	        // write -> global status
	        // Line A1
	        IF #Active.Line.A1 THEN
	            DB_Global.Status.Line.A1.On[#TransferID] := #ReadTransferStatus.ON;
	            DB_Global.Status.Line.A1.ReadyToRun[#TransferID] := #ReadTransferStatus.ReadytoRun;
	            DB_Global.Status.Line.A1.Occupied[#TransferID] := #ReadTransferStatus.Occupied;
	            DB_Global.Status.Line.A1.Running[#TransferID] := #ReadTransferStatus.Running;
	            DB_Global.Status.Line.A1.Fault[#TransferID] := #ReadTransferStatus.Fault;
	            DB_Global.Status.Line.A1.Estop[#TransferID] := #ReadTransferStatus.Estop;
	            DB_Global.Status.Line.A1.Manual[#TransferID] := #ReadTransferStatus.Manual;
	            DB_Global.Status.Line.A1.Stop[#TransferID] := #ReadTransferStatus.Stop;
	            DB_Global.Status.Line.A1.Blockage[#TransferID] := #ReadTransferStatus.Blockage;
	        END_IF;
	        // Line B1
	        IF #Active.Line.B1 THEN
	            DB_Global.Status.Line.B1.On[#TransferID] := #ReadTransferStatus.ON;
	            DB_Global.Status.Line.B1.ReadyToRun[#TransferID] := #ReadTransferStatus.ReadytoRun;
	            DB_Global.Status.Line.B1.Occupied[#TransferID] := #ReadTransferStatus.Occupied;
	            DB_Global.Status.Line.B1.Running[#TransferID] := #ReadTransferStatus.Running;
	            DB_Global.Status.Line.B1.Fault[#TransferID] := #ReadTransferStatus.Fault;
	            DB_Global.Status.Line.B1.Estop[#TransferID] := #ReadTransferStatus.Estop;
	            DB_Global.Status.Line.B1.Manual[#TransferID] := #ReadTransferStatus.Manual;
	            DB_Global.Status.Line.B1.Stop[#TransferID] := #ReadTransferStatus.Stop;
	            DB_Global.Status.Line.B1.Blockage[#TransferID] := #ReadTransferStatus.Blockage;
	        END_IF;
	        // Line C1
	        IF #Active.Line.C1 THEN
	            DB_Global.Status.Line.C1.On[#TransferID] := #ReadTransferStatus.ON;
	            DB_Global.Status.Line.C1.ReadyToRun[#TransferID] := #ReadTransferStatus.ReadytoRun;
	            DB_Global.Status.Line.C1.Occupied[#TransferID] := #ReadTransferStatus.Occupied;
	            DB_Global.Status.Line.C1.Running[#TransferID] := #ReadTransferStatus.Running;
	            DB_Global.Status.Line.C1.Fault[#TransferID] := #ReadTransferStatus.Fault;
	            DB_Global.Status.Line.C1.Estop[#TransferID] := #ReadTransferStatus.Estop;
	            DB_Global.Status.Line.C1.Manual[#TransferID] := #ReadTransferStatus.Manual;
	            DB_Global.Status.Line.C1.Stop[#TransferID] := #ReadTransferStatus.Stop;
	            DB_Global.Status.Line.C1.Blockage[#TransferID] := #ReadTransferStatus.Blockage;
	        END_IF;
	        // Line D1
	        IF #Active.Line.D1 THEN
	            DB_Global.Status.Line.D1.On[#TransferID] := #ReadTransferStatus.ON;
	            DB_Global.Status.Line.D1.ReadyToRun[#TransferID] := #ReadTransferStatus.ReadytoRun;
	            DB_Global.Status.Line.D1.Occupied[#TransferID] := #ReadTransferStatus.Occupied;
	            DB_Global.Status.Line.D1.Running[#TransferID] := #ReadTransferStatus.Running;
	            DB_Global.Status.Line.D1.Fault[#TransferID] := #ReadTransferStatus.Fault;
	            DB_Global.Status.Line.D1.Estop[#TransferID] := #ReadTransferStatus.Estop;
	            DB_Global.Status.Line.D1.Manual[#TransferID] := #ReadTransferStatus.Manual;
	            DB_Global.Status.Line.D1.Stop[#TransferID] := #ReadTransferStatus.Stop;
	            DB_Global.Status.Line.D1.Blockage[#TransferID] := #ReadTransferStatus.Blockage;
	        END_IF;
	        
	    END_REGION
	    
	END_REGION
	
	REGION Transfer Logic
	    
	    REGION infeed receive condition
	        
	        // NegEdgeUpstream
	        #NegEdgeUpstream(CLK := #Upstream);
	        
	        // item will be send into the transfer section when there is no other item
	        
	        IF #ReadTransferStatus.ReadytoRun AND
	            #Upstream AND
	            NOT #ReadTransferStatus.Occupied THEN
	            #Transfer.RcvInfeed := TRUE;
	        END_IF;
	        
	        // receive infeed tag goes to FALSE when the item from the previous conveyor is completly out of the previous conveyor
	        IF NOT #Upstream(* #NegEdgeUpstream.Q *)THEN
	            #Transfer.RcvInfeed := FALSE;
	        END_IF;
	        
	        // Receive infeed
	        #Transfer.StartSignal := #Transfer.RcvInfeed;
	        
	    END_REGION
	    
	    REGION Transfer direction outputs
	        
	        IF NOT #EndSensor AND NOT #"Left/RightSensor" AND NOT #ReadTransferStatus.Running THEN
	            
	            #sTransferDirection := #TransferDirection;
	            
	        END_IF;
	        
	        // Transfer Straight
	        
	        IF #sTransferDirection.Straight THEN
	            
	            IF #ReadTransferStatus.ReadytoRun AND
	                NOT #Transfer.RcvInfeed AND
	                #ReadTransferStatus.Occupied AND
	                NOT #Downstream
	            THEN
	                #Transfer.Command_1 := TRUE;
	                #Transfer.Command_2 := TRUE;
	            END_IF;
	            
	        END_IF;
	        
	        // Transfer Right
	        
	        IF #sTransferDirection.toRight THEN
	            
	            IF #ReadTransferStatus.ReadytoRun AND
	                NOT #Transfer.RcvInfeed AND
	                #ReadTransferStatus.Occupied AND
	                NOT #Downstream
	            THEN
	                #Transfer.Command_1 := TRUE;
	                #Transfer.Command_2 := FALSE;
	            END_IF;
	            
	        END_IF;
	        
	        // Transfer Left
	        
	        IF #sTransferDirection.toLeft THEN
	            
	            IF #ReadTransferStatus.ReadytoRun AND
	                NOT #Transfer.RcvInfeed AND
	                #ReadTransferStatus.Occupied AND
	                NOT #Downstream
	            THEN
	                #Transfer.Command_1 := FALSE;
	                #Transfer.Command_2 := TRUE;
	            END_IF;
	            
	        END_IF;
	        
	    END_REGION
	    
	    REGION TRANSFER OFF
	        
	        // Transfer commands Off
	        
	        IF NOT #ReadTransferStatus.ReadytoRun OR
	            #Transfer.RcvInfeed OR
	            (#ReadTransferStatus.Occupied AND
	            #Downstream) OR
	            NOT #ReadTransferStatus.Occupied
	        THEN
	            #Transfer.Command_1 := FALSE;
	            #Transfer.Command_2 := FALSE;
	        END_IF;
	        
	    END_REGION
	    
	    REGION Write output
	        
	        // Static to output
	        
	        #StartSignal := #Transfer.StartSignal;
	        #Cmd1 := #Transfer.Command_1;
	        #Cmd2 := #Transfer.Command_2;
	        
	    END_REGION
	    
	END_REGION
	
	
	
	
	
END_FUNCTION_BLOCK
END_NAMESPACE

NAMESPACE LineA1
FUNCTION_BLOCK FB_GetDiag
{ S7_Optimized_Access := 'TRUE' ; Published := 'TRUE' }
VERSION : 0.1
   VAR_INPUT 
      HardwareID : HW_ANY;
   END_VAR

   VAR_OUTPUT 
      CommunicationErrorAlarm : Bool;
   END_VAR

   VAR 
      GetDiag { S7_SetPoint := 'False'} : _.Global.GetDiag;
      CheckOwnState : UInt := 5;
      CommunicationError : Bool;
   END_VAR


BEGIN
	// ==========================================================================================================================================
	// Company        : LogTech, s.r.o.
	// Created by     : Anton Vinoth Soundraraj
	// Block          : FB_GetDiag
	// Project        : LT-Lib-Block
	// ==========================================================================================================================================
	
	REGION Get_Diag
	    
	    #GetDiag.ReturnValue := GET_DIAG(MODE := #GetDiag.DiagMode,
	                                     LADDR := #HardwareID,
	                                     CNT_DIAG => #GetDiag.CountDiagDetail,
	                                     DIAG := #GetDiag.MyDiag);
	END_REGION
	
	REGION Communiation_Error
	    
	    IF #GetDiag.MyDiag.OwnState = #CheckOwnState THEN
	        #CommunicationErrorAlarm := TRUE;
	    ELSE
	        #CommunicationErrorAlarm := FALSE;
	    END_IF;
	    
	    IF #GetDiag.MyDiag.OwnState = #CheckOwnState THEN
	        #CommunicationError := TRUE;
	    ELSE
	        #CommunicationError := FALSE;
	    END_IF;
	    
	END_REGION
	
	
END_FUNCTION_BLOCK
END_NAMESPACE

NAMESPACE Global
FUNCTION_BLOCK FB_HardwareDiag
{ S7_Optimized_Access := 'TRUE' ; Published := 'TRUE' }
VERSION : 0.1
   VAR 
      ASi : _.LineA1.FB_GetDiag;
   END_VAR


BEGIN
	// ==========================================================================================================================================
	// Company        : LogTech, s.r.o.
	// Created by     : Anton Vinoth Soundraraj
	// Block          : FB_HardwareDiag
	// Project        : Lékarna DC Chrudim
	// Project number : 23-157
	// ==========================================================================================================================================
	
	(* REGION ASi
	    
	    #ASi(HardwareID              := _."bu-asi-gw~PN-IO",
	         CommunicationErrorAlarm => _.Global.DB_Alarm.HardDiag.ASi.%X0);
	    
	    
	END_REGION *)
	
	
	
	
END_FUNCTION_BLOCK
END_NAMESPACE

NAMESPACE Global
FUNCTION FC_AllKlaxon : Void
{ S7_Optimized_Access := 'TRUE' ; Published := 'TRUE' }
VERSION : 0.1

BEGIN
	// ==========================================================================================================================================
	// Company        : LogTech, s.r.o.
	// Created by     : Anton Vinoth Soundraraj
	// Block          : FB_HardwareDiag
	// Project        : Lékarna DC Chrudim
	// Project number : 23-157
	// ==========================================================================================================================================
	
	
END_FUNCTION
END_NAMESPACE

NAMESPACE LineA1
FUNCTION FC_Init : Void
{ S7_Optimized_Access := 'TRUE' ; Published := 'TRUE' }
VERSION : 0.1

BEGIN
	
	
	
	_.LineA1.IDB_LineA1."Conveyor_A1.1.1".MotorType."24v-ASi" := TRUE;
	
	
	
	
	
	
	
	
	
	
	
	
	
	
END_FUNCTION
END_NAMESPACE

NAMESPACE LineA1
FUNCTION_BLOCK FB_Interlock
{ S7_Optimized_Access := 'TRUE' ; Published := 'TRUE' }
VERSION : 0.1

BEGIN
END_FUNCTION_BLOCK
END_NAMESPACE

NAMESPACE LineA1
FUNCTION FC_Downstream : Void
{ S7_Optimized_Access := 'TRUE' ; Published := 'TRUE' }
VERSION : 0.1

BEGIN
END_FUNCTION
END_NAMESPACE

NAMESPACE LineA1
FUNCTION FC_Fault : Void
{ S7_Optimized_Access := 'TRUE' ; Published := 'TRUE' }
VERSION : 0.1

BEGIN
END_FUNCTION
END_NAMESPACE

NAMESPACE LineA1
FUNCTION FC_Upstream : Void
{ S7_Optimized_Access := 'TRUE' ; Published := 'TRUE' }
VERSION : 0.1

BEGIN
END_FUNCTION
END_NAMESPACE

NAMESPACE LineA1
FUNCTION FC_Alarm : Void
{ S7_Optimized_Access := 'TRUE' ; Published := 'TRUE' }
VERSION : 0.1

BEGIN
END_FUNCTION
END_NAMESPACE

NAMESPACE LineA1
FUNCTION FC_SimuAlarm : Void
{ S7_Optimized_Access := 'TRUE' ; Published := 'FALSE' }
VERSION : 0.1

BEGIN
END_FUNCTION
END_NAMESPACE

NAMESPACE LineB1
FUNCTION_BLOCK FB_S300_FullControl
{ S7_Optimized_Access := 'TRUE' ; Published := 'TRUE' }
VERSION : 0.1
   VAR_INPUT 
      TransferID : Int;
      TransferSensor : Bool;
      BeltUp : Bool;
      RollerUp : Bool;
      Fault : Bool;
      ReadyToRCV : Bool;
      UpstreamStraight : Bool;
      UpstreamArm : Bool;
      FrontSensor : Bool;
      EndSensor : Bool;
      "Left/RightSensor" : Bool;
      Downstream : Bool;
      PriorityStraight : Bool;
      PriorityArm : Bool;
      FrontSensorFilterTime : Array[1..2] of Time;
   END_VAR

   VAR_OUTPUT 
      Direction : Bool;
      Cmd1 : Bool;
      Cmd2 : Bool;
      ErrorReset : Bool;
   END_VAR

   VAR 
      ReadInputSignal : Struct
         EmergencyStop : Bool;
         FireActive : Bool;
         Fault : Bool;
         TransferSensor : Bool;
      END_STRUCT;
      Active : Struct
         Line : Struct
            B1 : Bool;
         END_STRUCT;
      END_STRUCT;
      TRANSFER_SENSOR : _.Global.FB_Sensor;
      FRONT_SENSOR_FILTER : _.Global.FB_Sensor;
      TRANSFER_SENSOR_BLOCKAGE {InstructionName := 'TON_TIME'; LibVersion := '1.0'} : TON_TIME;
      FRONT_SENSOR_BLOCKAGE {InstructionName := 'TON_TIME'; LibVersion := '1.0'} : TON_TIME;
      END_SENSOR_BLOCKAGE {InstructionName := 'TON_TIME'; LibVersion := '1.0'} : TON_TIME;
      "LEFT/RIGHT_SENSOR_BLOCKAGE" {InstructionName := 'TON_TIME'; LibVersion := '1.0'} : TON_TIME;
      TRANSFER_STATUS_ON : _.Global.FB_StatusON;
      TRANSFER_STATUS_READY : _.Global.FB_StatusReady;
      TRANSFER_STATUS_FAULT : _.Global.FB_StatusFault;
      AUTO_RESET : _.Global.FB_AutoReset;
      StartUpTimer {InstructionName := 'TOF_TIME'; LibVersion := '1.0'; S7_SetPoint := 'False'} : TOF_TIME;
      FT_StartUp {InstructionName := 'F_TRIG'; LibVersion := '1.0'} : F_TRIG;
      SetStartUp { S7_SetPoint := 'True'} : Bool;
      Init : Struct
         Line : Struct
            A1 : String := 'LineA1';
         END_STRUCT;
      END_STRUCT;
      SSR : _.Global.SystemSSR;
      ReadTransferStatus : _.Global.ConveyorStatus;
      ReadTransferParameters : _.Global.ConveyorParameters := ((), [2(T#10ms)], (), (), ());
      ConveyorFault : _.Global.Fault;
      StartupTransfer { S7_SetPoint := 'True'} : Bool;
      FilteredSensor { S7_SetPoint := 'True'} : Bool;
      StopSystemFireActive : Bool;
      ClearTransferArea : Bool;
      AutoReset : Bool;
      VisuColor : Word;
      Transfer : Struct
         ErrorReset : Bool;
         Direction : Bool;
         Command_1 : Bool;
         Command_2 : Bool;
      END_STRUCT;
   END_VAR


BEGIN
	// ==========================================================================================================================================
	// Company        : LogTech, s.r.o.
	// Created by     : Anton Vinoth Soundraraj
	// Block          : FB_S300_tTransMode
	// Project        : Lékarna DC Chrudim
	// Project number : 23-157
	// ==========================================================================================================================================
	
	REGION Active Line
	    
	        #Active.Line.B1 := TRUE;
	        
	END_REGION
	
	REGION SystemSSR
	    
	    // Line B1
	    IF #Active.Line.B1 THEN
	        #SSR.StartSystem := _.Global.DB_SystemSSR.Line.B1.StartSystem;
	        #SSR.StopSystem := _.Global.DB_SystemSSR.Line.B1.StopSystem;
	        #SSR.ResetSystem := _.Global.DB_SystemSSR.Line.B1.ResetSystem;
	    END_IF;
	    
	END_REGION
	
	REGION Read Input
	    
	    // read all inputs to the block
	    // Conveyor input read signals
	    #ReadInputSignal.TransferSensor := #TransferSensor;
	    #ReadInputSignal.Fault := #Fault;
	    // Read static tag connections
	    #ReadInputSignal.EmergencyStop := // all estop zones are connected together
	    _.DB_SafetyStandard.ToStandard.EstopActive;
	    // Common system input Read
	    #ReadInputSignal.FireActive :=
	    _.Global.DB_SystemSimu.Fire; // simu call
	    
	END_REGION
	
	REGION Conveyor startup
	    
	    // Conveyor StartUp: Conveyor startup signal after preset time
	    #StartUpTimer.TOF(IN := #SSR.StartSystem,
	                      PT := #ReadTransferParameters.StartUpTime);
	    
	    #FT_StartUp(CLK := #StartUpTimer.Q);
	    
	    // set startup after the preset
	    #SetStartUp := #FT_StartUp.Q;
	    
	END_REGION
	
	REGION READ AND INIT
	    
	    REGION Init conveyor parameters
	        
	        // Conveyor Parameter
	        // Line B1
	        IF #Active.Line.B1 THEN
	            #ReadTransferParameters := DB_ConveyorParameters.Line.B1.Conveyor[#TransferID];
	        END_IF;
	        
	    END_REGION
	    
	    REGION Sensor Filter
	        
	        // FB_Sensor
	        // called as MIDB
	        
	        #TRANSFER_SENSOR(Sensor := #ReadInputSignal.TransferSensor,
	                         SensorFilterTime := #ReadTransferParameters.SensorFilterTime,
	                         FilteredSensor => #FilteredSensor);
	        
	        // front sensor filter
	        #FRONT_SENSOR_FILTER(Sensor := #FrontSensor,
	                             SensorFilterTime := #FrontSensorFilterTime);
	        
	    END_REGION
	    
	    REGION FIRE
	        
	        // Fire signal from fire system stops the whole system
	        // System can be reset from Fire status only if the fire signal is deactivated
	        
	        // FIRE ALARM ACTIVE --> STOP SYSTEM
	        IF #ReadInputSignal.FireActive THEN
	            #StopSystemFireActive := TRUE;
	        END_IF;
	        // RESET --> FIRE ALARM
	        IF #SSR.ResetSystem AND NOT #ReadInputSignal.FireActive THEN
	            #StopSystemFireActive := FALSE;
	        END_IF;
	        
	    END_REGION
	    
	END_REGION
	
	REGION Conveyor Status
	    
	    REGION Status ON
	        
	        // ----------------------------------------->>>>>>> STATUS ON <<<<<<<-----------------------------------------
	        // FB_ConveyorStatusON
	        // called as IDMB
	        
	        #TRANSFER_STATUS_ON(SystemStartActive := #SSR.StartSystem,
	                            StatusStop := #ReadTransferStatus.Stop,
	                            StatusEStop := #ReadTransferStatus.Estop,
	                            StatusManual := #ReadTransferStatus.Manual,
	                            StatusFault := #ReadTransferStatus.Fault,
	                            FireAlarmActive := #StopSystemFireActive,
	                            StatusON => #ReadTransferStatus.ON);
	        
	    END_REGION
	    
	    REGION Status Ready
	        
	        // ----------------------------------------->>>>>>> STATUS READY <<<<<<<-----------------------------------------
	        // FB_ConveyorStatusReady
	        // called as MIDB
	        
	        #TRANSFER_STATUS_READY(StatusON := #ReadTransferStatus.ON,
	                               StatusESTOP := #ReadTransferStatus.Estop,
	                               StatusFAULT := #ReadTransferStatus.Fault,
	                               StatusMAN := #ReadTransferStatus.Manual,
	                               SignalFIRE := #StopSystemFireActive,
	                               SystemAlertTime := #ReadTransferParameters.StartUpTime,
	                               StatusReady => #ReadTransferStatus.ReadytoRun);
	        
	    END_REGION
	    
	    REGION Status Occupied
	        
	        // ----------------------------------------->>>>>>> STATUS OCCUPIED <<<<<<<-----------------------------------------
	        
	        #ReadTransferStatus.Occupied :=
	        #FilteredSensor AND
	        NOT #FRONT_SENSOR_FILTER.FilteredSensor;
	        
	    END_REGION
	    
	    REGION Status Running
	        
	        // ----------------------------------------->>>>>>> STATUS RUNNING <<<<<<<-----------------------------------------
	        
	        #ReadTransferStatus.Running := #Transfer.Command_1 OR #Transfer.Command_2;
	        
	    END_REGION
	    
	    REGION Status Fault
	        
	        // Automatic reset trigger to the needed drive after wakeup from ESTOP power miss (only if needed)
	        // will trigger for every Reset active
	        
	        #AUTO_RESET(AckIN := #SSR.ResetSystem,
	                    Ack => #AutoReset);
	        
	        // ----------------------------------------->>>>>>> STATUS FAULT <<<<<<<-----------------------------------------
	        
	        #TRANSFER_STATUS_FAULT(FaultActive := #ReadInputSignal.Fault,
	                               ResetFault := #SSR.ResetSystem OR #AutoReset,
	                               StatusRunning := #ReadTransferStatus.Running,
	                               FaultStatus => #ReadTransferStatus.Fault);
	        
	        #ErrorReset := #SSR.ResetSystem AND #ReadTransferStatus.Fault;
	        
	    END_REGION
	    
	    REGION Status ESTOP
	        
	        // ----------------------------------------->>>>>>> STATUS ESTOP <<<<<<<-----------------------------------------
	        
	        // EMERGENCY STOP ACTIVE --> STOP SYSTEM
	        IF #ReadInputSignal.EmergencyStop THEN
	            #ReadTransferStatus.Estop := TRUE;
	        END_IF;
	        // RESET --> EMERGENCY STOP
	        IF #AutoReset AND NOT #ReadInputSignal.EmergencyStop THEN
	            #ReadTransferStatus.Estop := FALSE;
	        END_IF;
	        
	    END_REGION
	    
	    REGION Status Manual
	        
	        // ----------------------------------------->>>>>>> STATUS MANUAL <<<<<<<-----------------------------------------
	        
	        // Write to static from IO
	        // ACTIVATE --> MANUAL MODE
	        // Line B1
	        IF #Active.Line.B1 THEN
	            // SET --> MANUAL MODE
	            IF DB_Manual.Line.B1.Conveyor[#TransferID].ManualEnable THEN
	                #ReadTransferStatus.Manual := TRUE;
	            END_IF;
	            // RESET --> MANUAL MODE
	            IF NOT DB_Manual.Line.B1.Conveyor[#TransferID].ManualEnable AND #SSR.ResetSystem THEN
	                #ReadTransferStatus.Manual := FALSE;
	            END_IF;
	        END_IF;
	        
	    END_REGION
	    
	    REGION Status Stop
	        
	        // ----------------------------------------->>>>>>> STATUS STOP <<<<<<<-----------------------------------------
	        
	        IF #SSR.StopSystem THEN
	            #ReadTransferStatus.Stop := TRUE;
	        END_IF;
	        IF #SSR.StartSystem OR #SSR.ResetSystem THEN
	            #ReadTransferStatus.Stop := FALSE;
	        END_IF;
	        
	    END_REGION
	    
	    REGION Status Blockage
	        
	        // FB_SensorBlockage
	        // called as MIDB
	        #TRANSFER_SENSOR_BLOCKAGE(IN := #ReadTransferStatus.ReadytoRun AND #FilteredSensor AND NOT #Downstream,
	                                  PT := T#15s);
	        
	        #FRONT_SENSOR_BLOCKAGE(IN := #ReadTransferStatus.ReadytoRun AND #FrontSensor AND NOT #Downstream,
	                               PT := T#15s);
	        
	        #END_SENSOR_BLOCKAGE(IN := #ReadTransferStatus.ReadytoRun AND #EndSensor AND NOT #Downstream,
	                             PT := T#15s);
	        
	        #"LEFT/RIGHT_SENSOR_BLOCKAGE"(IN := #ReadTransferStatus.ReadytoRun AND #"Left/RightSensor" AND NOT #Downstream,
	                                      PT := T#5s);
	        
	        #ReadTransferStatus.Blockage :=
	        (#TRANSFER_SENSOR_BLOCKAGE.Q OR
	        #FRONT_SENSOR_BLOCKAGE.Q OR
	        #END_SENSOR_BLOCKAGE.Q OR
	        #"LEFT/RIGHT_SENSOR_BLOCKAGE".Q);
	        
	        // ==========================
	        // Sensor Blockage: HMI Alarm
	        // ==========================
	        // Sensor blockage alarm message is written to the alarm word
	        // corresponding to the active line
	        
	        REGION alarm 
	            
	            // ==========================
	            // Sensor Blockage: HMI Alarm
	            // ==========================
	            // Sensor blockage alarm message is written to the alarm word
	            // corresponding to the active line
	            // Line B1
	            IF #Active.Line.B1 THEN
	                DB_Alarm."word".Line.B1.Conveyor[#TransferID].%X0 := #ReadTransferStatus.Blockage;
	            END_IF;
	            
	        END_REGION
	        
	    END_REGION
	    
	    REGION Visu Color
	        
	        // each and every status of the conveyor will be mentioned by different colors in HMI panel
	        
	        #VisuColor.%X8 := #ReadTransferStatus.Blockage;
	        #VisuColor.%X0 := #ReadTransferStatus.ON;
	        #VisuColor.%X1 := #ReadTransferStatus.ReadytoRun;
	        #VisuColor.%X2 := #ReadTransferStatus.Occupied;
	        #VisuColor.%X3 := #ReadTransferStatus.Running;
	        #VisuColor.%X4 := #ReadTransferStatus.Fault;
	        #VisuColor.%X5 := #ReadTransferStatus.Estop;
	        #VisuColor.%X6 := #ReadTransferStatus.Manual;
	        #VisuColor.%X7 := #ReadTransferStatus.Stop;
	        
	        // convert word to Interger value: 
	        // color will be depends on the status priority (integer value) 
	        // reference: Conveyor image in HMI screen -> property -> Apperance   
	        
	        // Line B1
	        IF #Active.Line.B1 THEN
	            _.Global.DB_VisuColor.Line.B1.Conveyor[#TransferID] :=
	            WORD_TO_INT(#VisuColor);
	        END_IF;
	        
	    END_REGION
	    
	    REGION Global Status
	        
	        // write -> global status
	        // Line B1
	        IF #Active.Line.B1 THEN
	            _.Global.DB_Global.Status.Line.B1.On[#TransferID] := #ReadTransferStatus.ON;
	            _.Global.DB_Global.Status.Line.B1.ReadyToRun[#TransferID] := #ReadTransferStatus.ReadytoRun;
	            _.Global.DB_Global.Status.Line.B1.Occupied[#TransferID] := #ReadTransferStatus.Occupied;
	            _.Global.DB_Global.Status.Line.B1.Running[#TransferID] := #ReadTransferStatus.Running;
	            _.Global.DB_Global.Status.Line.B1.Fault[#TransferID] := #ReadTransferStatus.Fault;
	            _.Global.DB_Global.Status.Line.B1.Estop[#TransferID] := #ReadTransferStatus.Estop;
	            _.Global.DB_Global.Status.Line.B1.Manual[#TransferID] := #ReadTransferStatus.Manual;
	            _.Global.DB_Global.Status.Line.B1.Stop[#TransferID] := #ReadTransferStatus.Stop;
	            _.Global.DB_Global.Status.Line.B1.Blockage[#TransferID] := #ReadTransferStatus.Blockage;
	        END_IF;
	        
	    END_REGION
	    
	END_REGION
	
	REGION Transfer Logic
	    
	    IF #ReadTransferStatus.ReadytoRun THEN
	        
	        REGION Belt going UP
	            
	            // tote from straight has higher priority
	            // upstream straight is satisfied (add upstream sensor and front sensor)
	            // transfer is not occupied
	            // belt is not UP
	            IF (#PriorityStraight AND
	                #UpstreamStraight AND
	                NOT #ReadTransferStatus.Occupied AND
	                NOT #BeltUp) OR
	                // transfer has received an item from arm
	                // belt is not UP
	                (#ReadTransferStatus.Occupied AND
	                NOT #BeltUp)
	            THEN
	                #Transfer.Command_1 := TRUE;
	                #Transfer.Command_2 := TRUE;
	                #Transfer.Direction := TRUE;
	            END_IF;
	            
	        END_REGION
	        
	        REGION Roller going UP
	            
	            // tote from arm has higher priority
	            // upstream arm is satisfied (add upstream sensor and left/right sensor)
	            // transfer is not occupied
	            // roller is not UP
	            IF (#PriorityArm AND
	                #UpstreamArm AND
	                NOT #ReadTransferStatus.Occupied AND
	                NOT #RollerUp)
	            THEN
	                #Transfer.Command_1 := TRUE;
	                #Transfer.Command_2 := TRUE;
	                #Transfer.Direction := FALSE;
	            END_IF;
	            
	        END_REGION
	        
	        REGION Belt rcv and trs item
	            
	            IF // belt rcv the item (from straight)
	                (#BeltUp AND
	                NOT #ReadTransferStatus.Occupied AND
	                #PriorityStraight AND
	                #UpstreamStraight) OR
	                // belt trs the item
	                (#BeltUp AND
	                #ReadTransferStatus.Occupied AND
	                NOT #Downstream)
	            THEN
	                #Transfer.Command_1 := TRUE;
	                #Transfer.Command_2 := FALSE;
	                #Transfer.Direction := FALSE;
	            END_IF;
	            
	        END_REGION
	        
	    END_IF;
	    
	    REGION TRANSFER OFF
	        
	        IF NOT #ReadTransferStatus.ReadytoRun OR
	            (#ReadTransferStatus.Occupied AND
	            #Downstream)
	        THEN
	            #Transfer.Command_1 := FALSE;
	            #Transfer.Command_2 := FALSE;
	        END_IF;
	        
	    END_REGION
	    
	    REGION Write output
	        
	        // Static to output
	        
	        #Direction := #Transfer.Direction;
	        #Cmd1 := #Transfer.Command_1;
	        #Cmd2 := #Transfer.Command_2;
	        #ErrorReset := #Transfer.ErrorReset;
	        
	    END_REGION
	    
	END_REGION
	
	
	
	
	
END_FUNCTION_BLOCK
END_NAMESPACE

NAMESPACE Global
FUNCTION_BLOCK FB_MABS_Profinet
{ S7_Optimized_Access := 'TRUE' ; Published := 'TRUE' }
VERSION : 0.1
   VAR_INPUT 
      MABS_ID : Int;
      CrossSensor : Bool;
      Fault : Bool;
      UpstreamRunning : Bool;
      Downstream_Straight : Bool;
      "Downstream_Right/Left" : Bool;
      SortDir : ItemDir;
      ManIn : MABS_ManIn;
      Setpoints : MABS_Setpoint;
   END_VAR

   VAR_IN_OUT 
      MABS_IBP_in : IB_P01_02_03_in_64bytes_struct;
      MABS_IBP_out : IB_P01_02_03_out_64bytes_struct;
   END_VAR

   VAR 
      ReadInputSignal : Struct
         CrossSensor : Bool;
         EmergencyStop : Bool;
         Fault : Bool;
      END_STRUCT;
      Active : Struct
         Line : Struct
            ProductionLine : Bool;
            EmptyLine : Bool;
            PackedLine : Bool;
         END_STRUCT;
         EstopZone { S7_SetPoint := 'False'} : EsopZone;
      END_STRUCT;
      CROSS_SENSOR_FILTER : FB_Sensor;
      MABS_SENSOR_BLOCKAGE {InstructionName := 'IEC_TIMER'; LibVersion := '1.0'} : IEC_TIMER;
      MABS_STATUS_ON : FB_StatusON;
      MABS_STATUS_READY : FB_StatusReady;
      MABS_STATUS_FAULT : FB_StatusFault;
      AUTO_RESET : FB_AutoReset;
      MABS_CONTROL : FB_MABS_PNIO;
      SSR : SystemSSR;
      ReadMabsStatus : ConveyorStatus;
      ReadMabsParameter : ConveyorParameters := ((), [2(T#10ms)], (), (), (), ());
      MABSFault : Fault;
      SimuMode : Struct
         Sensor : Bool;
         Fault : Bool;
      END_STRUCT;
      StartUpTimer {InstructionName := 'TOF_TIME'; LibVersion := '1.0'; S7_SetPoint := 'False'} : TOF_TIME;
      FT_StartUp {InstructionName := 'F_TRIG'; LibVersion := '1.0'} : F_TRIG;
      SetStartUp { S7_SetPoint := 'True'} : Bool;
      VisuColor : Word;
      PhaseError : Bool;
      StartupMABS { S7_SetPoint := 'True'} : Bool;
      FilteredSensor { S7_SetPoint := 'True'} : Bool;
      AutoReset { S7_SetPoint := 'True'} : Bool;
      StopSystemFireActive : Bool;
      Sort { S7_SetPoint := 'False'} : ItemDir;
      Home : Bool;
      HomeCheckTimer {InstructionName := 'TON_TIME'; LibVersion := '1.0'} : TON_TIME;
      CurrentPosition : Struct
         left : Bool;
         right : Bool;
         straight : Bool;
      END_STRUCT;
      "Cmd+Setpoint" { ExternalAccessible := 'False'; ExternalVisible := 'False'; ExternalWritable := 'False'; S7_SetPoint := 'False'} : MABS;
   END_VAR


BEGIN
	// ==========================================================================================================================================
	// Company        : LogTech, s.r.o.
	// Created by     : Anton Vinoth Soundraraj
	// Block          : FB_MABS
	// Project        : Lékarna DC Chrudim
	// Project number : 23-157
	// ==========================================================================================================================================
	
	REGION Active Line
	    
	    // ProductionLine
	    IF (#MABS_ID >= _.gminProductionLine AND
	        #MABS_ID <= _.gmaxProductionLine)
	    THEN
	        #Active.Line.ProductionLine := TRUE;
	    END_IF;
	    
	    // EmptyLine
	    IF (#MABS_ID >= _.gminEmptyLine AND
	        #MABS_ID <= _.gmaxEmptyLine)
	    THEN
	        #Active.Line.EmptyLine := TRUE;
	    END_IF;
	    
	    // PackedLine
	    IF (#MABS_ID >= _.gminPackedLine AND
	        #MABS_ID <= _.gmaxPackedLine)
	    THEN
	        #Active.Line.PackedLine := TRUE;
	    END_IF;
	    
	END_REGION
	
	REGION Estop zone
	    
	    // Production Line A1
	    IF  (#MABS_ID >= _."gA1.6.1" AND
	        #MABS_ID <= _."gA1.6.2") OR
	        // Empty Line A1
	        (#MABS_ID >= _."gJ1.5.2" AND
	        #MABS_ID <= _."gJ1.6.2")
	    THEN
	        #Active.EstopZone."1" := TRUE;
	    END_IF;
	    
	    // Production Line A2
	    IF  (#MABS_ID >= _."gA1.9.1" AND
	        #MABS_ID <= _."gA1.9.2")
	    THEN
	        #Active.EstopZone."2" := TRUE;
	    END_IF;
	    
	END_REGION
	
	REGION SystemSSR
	    
	    //Zone 1
	    IF #Active.EstopZone."1" THEN
	        #SSR.StartSystem := DB_SystemSSR.Zone."1".StartSystem;
	        #SSR.StopSystem := DB_SystemSSR.Zone."1".StopSystem;
	        #SSR.ResetSystem := DB_SystemSSR.Zone."1".ResetSystem;
	    END_IF;
	    
	    //Zone 2
	    IF #Active.EstopZone."2" THEN
	        #SSR.StartSystem := DB_SystemSSR.Zone."2".StartSystem;
	        #SSR.StopSystem := DB_SystemSSR.Zone."2".StopSystem;
	        #SSR.ResetSystem := DB_SystemSSR.Zone."2".ResetSystem;
	    END_IF;
	    
	END_REGION
	
	REGION Read Simu inputs  
	    
	    // ProductionLine
	    IF #Active.Line.ProductionLine THEN
	        // read simu
	        #SimuMode.Sensor := DB_SystemSimu.TriggerSensor.Line.ProductionLine.Conveyor[#MABS_ID];
	        #SimuMode.Fault := DB_SystemSimu.TriggerFault.Line.ProductionLine.Conveyor[#MABS_ID];
	    END_IF;
	    
	    // EmptyLine
	    IF #Active.Line.EmptyLine THEN
	        // read simu
	        #SimuMode.Sensor := DB_SystemSimu.TriggerSensor.Line.EmptyLine.Conveyor[#MABS_ID];
	        #SimuMode.Fault := DB_SystemSimu.TriggerFault.Line.EmptyLine.Conveyor[#MABS_ID];
	    END_IF;
	    
	    // PackedLine
	    IF #Active.Line.PackedLine THEN
	        // read simu
	        #SimuMode.Sensor := DB_SystemSimu.TriggerSensor.Line.PackedLine.Conveyor[#MABS_ID];
	        #SimuMode.Fault := DB_SystemSimu.TriggerFault.Line.PackedLine.Conveyor[#MABS_ID];
	    END_IF;
	    
	END_REGION
	
	REGION Read Input
	    
	    // read all inputs to the block
	    // Conveyor input read signals
	    #ReadInputSignal.CrossSensor := #CrossSensor OR  // Not
	    #SimuMode.Sensor; // simu call
	    #ReadInputSignal.Fault := #Fault OR
	    #SimuMode.Fault; // simu call;
	    #ReadInputSignal.EmergencyStop := // all estop zones are connected together
	    _.DB_SafetyStandard.ToStandard.EstopActive;
	    
	END_REGION
	
	REGION READ AND INIT
	    
	    REGION parameters
	        
	        // ProductionLine
	        IF #Active.Line.ProductionLine THEN
	            #ReadMabsParameter := DB_ConveyorParameters.Line.ProductionLine.Conveyor[#MABS_ID];
	        END_IF;
	        // EmptyLine
	        IF #Active.Line.EmptyLine THEN
	            #ReadMabsParameter := DB_ConveyorParameters.Line.EmptyLine.Conveyor[#MABS_ID];
	        END_IF;
	        // PackedLine
	        IF #Active.Line.PackedLine THEN
	            #ReadMabsParameter := DB_ConveyorParameters.Line.PackedLine.Conveyor[#MABS_ID];
	        END_IF;
	        
	    END_REGION
	    
	    REGION FIRE
	        
	        // Fire signal from fire system stops the whole system
	        // System can be reset from Fire status only if the fire signal is deactivated
	        
	        // FIRE ALARM ACTIVE --> STOP SYSTEM
	        IF DB_SystemSimu.Fire THEN
	            #StopSystemFireActive := TRUE;
	        END_IF;
	        // RESET --> FIRE ALARM
	        IF #SSR.ResetSystem AND NOT DB_SystemSimu.Fire THEN
	            #StopSystemFireActive := FALSE;
	        END_IF;
	        
	    END_REGION
	    
	END_REGION
	
	REGION Conveyor startup
	    
	    // Conveyor StartUp: Conveyor startup signal after 5 second delay
	    
	    #StartUpTimer.TOF(IN := #SSR.StartSystem,
	                      PT := #ReadMabsParameter.StartUpTime);
	    
	    #FT_StartUp(CLK := #StartUpTimer.Q);
	    
	    // set startup after 5 seconds
	    #SetStartUp := #FT_StartUp.Q;
	    
	END_REGION
	
	REGION Conveyor Status
	    
	    REGION Status ON
	        
	        // ----------------------------------------->>>>>>> STATUS ON <<<<<<<-----------------------------------------
	        // FB_ConveyorStatusON
	        // called as IDMB
	        
	        #MABS_STATUS_ON(SystemStartActive := #SSR.StartSystem,
	                        StatusStop := #ReadMabsStatus.Stop,
	                        StatusEStop := #ReadMabsStatus.Estop,
	                        StatusManual := #ReadMabsStatus.Manual,
	                        StatusFault := #ReadMabsStatus.Fault,
	                        FireAlarmActive := #StopSystemFireActive,
	                        StatusON => #ReadMabsStatus.ON);
	        
	    END_REGION
	    
	    REGION Status Ready
	        
	        // ----------------------------------------->>>>>>> STATUS READY <<<<<<<-----------------------------------------
	        // FB_ConveyorStatusReady
	        // called as MIDB
	        
	        #MABS_STATUS_READY(StatusON := #ReadMabsStatus.ON,
	                           StatusESTOP := #ReadMabsStatus.Estop,
	                           StatusFAULT := #ReadMabsStatus.Fault,
	                           StatusMAN := #ReadMabsStatus.Manual,
	                           SignalFIRE := #StopSystemFireActive,
	                           SystemAlertTime := #ReadMabsParameter.StartUpTime,
	                           StatusReady => #ReadMabsStatus.ReadytoRun);
	        
	    END_REGION
	    
	    REGION Status Occupied
	        
	        // ----------------------------------------->>>>>>> STATUS OCCUPIED <<<<<<<-----------------------------------------
	        
	        #ReadMabsStatus.Occupied :=
	        #CROSS_SENSOR_FILTER.FilteredSensor;
	        
	    END_REGION
	    
	    REGION Status Running
	        
	        // ----------------------------------------->>>>>>> STATUS RUNNING <<<<<<<-----------------------------------------
	        
	        #ReadMabsStatus.Running :=
	        #ReadMabsStatus.ReadytoRun AND
	        #"Cmd+Setpoint".Run_balls;
	        
	    END_REGION
	    
	    REGION Status Fault
	        
	        // ----------------------------------------->>>>>>> STATUS FAULT <<<<<<<-----------------------------------------
	        
	        // Reading error signal from the motor drive
	        #MABSFault.Motor_Error := #ReadInputSignal.Fault;
	        
	        // FC_ConveyorStatusFault
	        #MABS_STATUS_FAULT(FaultActive := #MABSFault.Motor_Error,
	                           ResetFault := #SSR.ResetSystem,
	                           StatusRunning := #ReadMabsStatus.Running,
	                           FaultStatus => #ReadMabsStatus.Fault);
	        
	    END_REGION
	    
	    REGION Status ESTOP
	        
	        // ----------------------------------------->>>>>>> STATUS ESTOP <<<<<<<-----------------------------------------
	        
	        #AUTO_RESET(AckIN := #SSR.ResetSystem,
	                    Ack => #AutoReset);
	        
	        // EMERGENCY STOP ACTIVE --> STOP SYSTEM
	        IF #ReadInputSignal.EmergencyStop THEN
	            #ReadMabsStatus.Estop := TRUE;
	        END_IF;
	        // RESET --> EMERGENCY STOP
	        IF #AutoReset AND NOT #ReadInputSignal.EmergencyStop THEN
	            #ReadMabsStatus.Estop := FALSE;
	        END_IF;
	        
	    END_REGION
	    
	    REGION Status Stop
	        
	        // ----------------------------------------->>>>>>> STATUS STOP <<<<<<<-----------------------------------------
	        
	        IF #SSR.StopSystem THEN
	            #ReadMabsStatus.Stop := TRUE;
	        END_IF;
	        IF #SSR.StartSystem OR #SSR.ResetSystem THEN
	            #ReadMabsStatus.Stop := FALSE;
	        END_IF;
	        
	    END_REGION
	    
	    REGION Sensor Blockage
	        
	        // ----------------------------------------->>>>>>> STATUS BLOCKAGE <<<<<<<-------------------------------------
	        
	        // FB_SensorBlockage
	        // called as MIDB
	        
	        #MABS_SENSOR_BLOCKAGE.TON(IN := #ReadMabsStatus.ReadytoRun AND
	                                  #CROSS_SENSOR_FILTER.FilteredSensor,
	                                  PT := #ReadMabsParameter.SensorBlockageTime,
	                                  Q => #ReadMabsStatus.Blockage);
	        
	        // ==========================
	        // Sensor Blockage: HMI Alarm
	        // ==========================
	        // Sensor blockage alarm message is written to the first bit of the alarm word
	        // corresponding to the active line
	        
	        REGION alarm 
	            
	            // ==========================
	            // Sensor Blockage: HMI Alarm
	            // ==========================
	            // Sensor blockage alarm message is written to the alarm word
	            // corresponding to the active line
	            // ProductionLine
	            IF #Active.Line.ProductionLine THEN
	                DB_Alarm."word".Line.ProductionLine.Conveyor[#MABS_ID].%X0 := #ReadMabsStatus.Blockage;
	            END_IF;
	            // EmptyLine
	            IF #Active.Line.EmptyLine THEN
	               DB_Alarm."word".Line.EmptyLine.Conveyor[#MABS_ID].%X0 := #ReadMabsStatus.Blockage;
	            END_IF;
	            // PackedLine
	            IF #Active.Line.PackedLine THEN
	               DB_Alarm."word".Line.PackedLine.Conveyor[#MABS_ID].%X0 := #ReadMabsStatus.Blockage;
	            END_IF;
	            
	        END_REGION
	        
	    END_REGION
	    
	    REGION Visu Color
	        
	        // each and every status of the conveyor will be mentioned by different colors in HMI panel
	        
	        #VisuColor.%X8 := #ReadMabsStatus.Blockage;
	        #VisuColor.%X0 := #ReadMabsStatus.ON;
	        #VisuColor.%X1 := #ReadMabsStatus.ReadytoRun;
	        #VisuColor.%X2 := #ReadMabsStatus.Occupied;
	        #VisuColor.%X3 := #ReadMabsStatus.Running;
	        #VisuColor.%X4 := #ReadMabsStatus.Fault;
	        #VisuColor.%X5 := #ReadMabsStatus.Estop;
	        #VisuColor.%X6 := #ReadMabsStatus.Manual;
	        #VisuColor.%X7 := #ReadMabsStatus.Stop;
	        
	        // convert word to Interger value: 
	        // color will be depends on the status priority (integer value) 
	        // reference: Conveyor image in HMI screen -> property -> Apperance   
	        
	        // ProductionLine
	        IF #Active.Line.ProductionLine THEN
	            DB_VisuColor.Line.ProductionLine.Conveyor[#MABS_ID] :=
	            WORD_TO_INT(#VisuColor);
	        END_IF;
	        // EmptyLine
	        IF #Active.Line.EmptyLine THEN
	            DB_VisuColor.Line.EmptyLine.Conveyor[#MABS_ID] :=
	            WORD_TO_INT(#VisuColor);
	        END_IF;
	        // PackedLine
	        IF #Active.Line.PackedLine THEN
	            DB_VisuColor.Line.PackedLine.Conveyor[#MABS_ID] :=
	            WORD_TO_INT(#VisuColor);
	        END_IF;
	        
	    END_REGION
	    
	    REGION Global Status
	        
	        // write -> global status
	        // ProductionLine
	        IF #Active.Line.ProductionLine THEN
	            DB_Global.Status.Line.ProductionLine.On[#MABS_ID] := #ReadMabsStatus.ON;
	            DB_Global.Status.Line.ProductionLine.ReadyToRun[#MABS_ID] := #ReadMabsStatus.ReadytoRun;
	            DB_Global.Status.Line.ProductionLine.Occupied[#MABS_ID] := #ReadMabsStatus.Occupied;
	            DB_Global.Status.Line.ProductionLine.Running[#MABS_ID] := #ReadMabsStatus.Running;
	            DB_Global.Status.Line.ProductionLine.Fault[#MABS_ID] := #ReadMabsStatus.Fault;
	            DB_Global.Status.Line.ProductionLine.Estop[#MABS_ID] := #ReadMabsStatus.Estop;
	            DB_Global.Status.Line.ProductionLine.Manual[#MABS_ID] := #ReadMabsStatus.Manual;
	            DB_Global.Status.Line.ProductionLine.Stop[#MABS_ID] := #ReadMabsStatus.Stop;
	            DB_Global.Status.Line.ProductionLine.Blockage[#MABS_ID] := #ReadMabsStatus.Blockage;
	        END_IF;
	        // EmptyLine
	        IF #Active.Line.EmptyLine THEN
	            DB_Global.Status.Line.EmptyLine.On[#MABS_ID] := #ReadMabsStatus.ON;
	            DB_Global.Status.Line.EmptyLine.ReadyToRun[#MABS_ID] := #ReadMabsStatus.ReadytoRun;
	            DB_Global.Status.Line.EmptyLine.Occupied[#MABS_ID] := #ReadMabsStatus.Occupied;
	            DB_Global.Status.Line.EmptyLine.Running[#MABS_ID] := #ReadMabsStatus.Running;
	            DB_Global.Status.Line.EmptyLine.Fault[#MABS_ID] := #ReadMabsStatus.Fault;
	            DB_Global.Status.Line.EmptyLine.Estop[#MABS_ID] := #ReadMabsStatus.Estop;
	            DB_Global.Status.Line.EmptyLine.Manual[#MABS_ID] := #ReadMabsStatus.Manual;
	            DB_Global.Status.Line.EmptyLine.Stop[#MABS_ID] := #ReadMabsStatus.Stop;
	            DB_Global.Status.Line.EmptyLine.Blockage[#MABS_ID] := #ReadMabsStatus.Blockage;
	        END_IF;
	        // PackedLine
	        IF #Active.Line.PackedLine THEN
	            DB_Global.Status.Line.PackedLine.On[#MABS_ID] := #ReadMabsStatus.ON;
	            DB_Global.Status.Line.PackedLine.ReadyToRun[#MABS_ID] := #ReadMabsStatus.ReadytoRun;
	            DB_Global.Status.Line.PackedLine.Occupied[#MABS_ID] := #ReadMabsStatus.Occupied;
	            DB_Global.Status.Line.PackedLine.Running[#MABS_ID] := #ReadMabsStatus.Running;
	            DB_Global.Status.Line.PackedLine.Fault[#MABS_ID] := #ReadMabsStatus.Fault;
	            DB_Global.Status.Line.PackedLine.Estop[#MABS_ID] := #ReadMabsStatus.Estop;
	            DB_Global.Status.Line.PackedLine.Manual[#MABS_ID] := #ReadMabsStatus.Manual;
	            DB_Global.Status.Line.PackedLine.Stop[#MABS_ID] := #ReadMabsStatus.Stop;
	            DB_Global.Status.Line.PackedLine.Blockage[#MABS_ID] := #ReadMabsStatus.Blockage;
	        END_IF;
	        
	    END_REGION
	    
	END_REGION
	
	REGION Sorter sensor filter
	    
	    // cross sensor filter
	    #CROSS_SENSOR_FILTER(Sensor :=  #ReadInputSignal.CrossSensor,   ///#CrossSensor
	                         SensorFilterTime := #ReadMabsParameter.SensorFilterTime,
	                         FilteredSensor=> #FilteredSensor);
	    
	END_REGION
	
	REGION MABS LOGIC
	    
	    REGION rcv direction 
	        
	        IF NOT #FilteredSensor THEN
	            #Sort := #SortDir;
	        END_IF;
	        
	    END_REGION
	    
	    REGION MABS lib block
	        
	        #MABS_CONTROL(IBP_in  := #MABS_IBP_in,
	                      IBP_out := #MABS_IBP_out,
	                      MABS    := #"Cmd+Setpoint");
	        
	    END_REGION
	    
	    REGION run MABS wheels
	        
	        #"Cmd+Setpoint".Run_balls := #UpstreamRunning;
	        
	    END_REGION
	    
	    REGION Current position
	        
	        #CurrentPosition.left := #"Cmd+Setpoint".Left_Pos_reach;
	        #CurrentPosition.right := #"Cmd+Setpoint".Right_Pos_reach;
	        #CurrentPosition.straight := #"Cmd+Setpoint".Straight_Pos_reach;
	        
	    END_REGION
	    
	    REGION HOMING
	        
	        // ==========================================================================================================================
	        // Initial operation (home searching)
	        // ==================================
	        
	        // Home missing (if MABS could not receive any position in 't' duration)
	        #HomeCheckTimer.TON(IN := NOT #CurrentPosition.left AND
	                            NOT #CurrentPosition.right AND
	                            NOT #CurrentPosition.straight,
	                            PT := T#2s);
	        #Home :=
	        NOT #HomeCheckTimer.Q;
	        
	        // init HOME
	        IF NOT #Home AND NOT #ReadMabsStatus.Stop THEN
	            #"Cmd+Setpoint".Init := TRUE;
	        END_IF;
	        // RESET -> Init Home
	        IF #Home THEN
	            #"Cmd+Setpoint".Init := TRUE;
	        END_IF;
	        
	    END_REGION
	    
	    REGION Parameters
	        
	        // change balls direction
	        #"Cmd+Setpoint".Dir_balls := #Setpoints.ChangeBallsDirection;
	        // balls speed
	        #"Cmd+Setpoint".Speed_balls := #Setpoints.Speed_balls;
	        // offset for straight
	        #"Cmd+Setpoint".Init_offset := #Setpoints.Init_offset;
	        
	    END_REGION
	    
	    REGION Sorting logic
	        
	        IF #ReadMabsStatus.ReadytoRun
	        THEN
	            
	            REGION Straight
	                
	                // ================================================== ^^^
	                
	                // sort straight - actual position: right
	                
	                IF #Sort.Straight AND
	                    NOT #CurrentPosition.straight AND
	                    #CurrentPosition.right AND
	                    NOT #CROSS_SENSOR_FILTER.FilteredSensor
	                THEN
	                    #"Cmd+Setpoint".Switch_right_to_st := TRUE;
	                ELSE
	                    #"Cmd+Setpoint".Switch_right_to_st := FALSE;
	                END_IF;
	                
	                // sort straight - actual position: left
	                
	                IF #Sort.Straight AND
	                    NOT #CurrentPosition.straight AND
	                    #CurrentPosition.left AND
	                    NOT #CROSS_SENSOR_FILTER.FilteredSensor
	                THEN
	                    #"Cmd+Setpoint".Switch_left_to_st := TRUE;
	                ELSE
	                    #"Cmd+Setpoint".Switch_left_to_st := FALSE;
	                END_IF;
	                
	            END_REGION
	            
	            REGION to Right
	                
	                // ================================================== >>>
	                
	                // sort right - actual position: straight/left
	                
	                IF #Sort.toRight AND
	                    NOT #CurrentPosition.right AND
	                    (#CurrentPosition.straight OR
	                    #CurrentPosition.left) AND
	                    NOT #CROSS_SENSOR_FILTER.FilteredSensor
	                THEN
	                    #"Cmd+Setpoint".Switch_right := TRUE;
	                ELSE
	                    #"Cmd+Setpoint".Switch_right := FALSE;
	                END_IF;
	                
	            END_REGION
	            
	            REGION to left
	                
	                // ================================================== <<<
	                
	                // sort left - actual position: straight/right
	                
	                IF #Sort.toLeft AND
	                    NOT #CurrentPosition.left AND
	                    (#CurrentPosition.straight OR
	                    #CurrentPosition.right) AND
	                    NOT #CROSS_SENSOR_FILTER.FilteredSensor
	                THEN
	                    #"Cmd+Setpoint".Switch_left := TRUE;
	                ELSE
	                    #"Cmd+Setpoint".Switch_left := FALSE;
	                END_IF;
	                
	            END_REGION
	            
	            // ============================================================================================================
	            
	        END_IF;
	        
	    END_REGION
	    
	   REGION reset error 
	        
	        // reset error
	       IF #ReadMabsStatus.Fault AND
	           #SSR.ResetSystem
	       THEN
	            #"Cmd+Setpoint".Reset_error := TRUE;
	        ELSE
	            #"Cmd+Setpoint".Reset_error := FALSE;
	        END_IF;
	        
	    END_REGION
	    
	    REGION stop function
	        
	        // stop if not ready
	        IF NOT #ReadMabsStatus.ReadytoRun AND NOT #ReadMabsStatus.Manual
	        THEN
	            #"Cmd+Setpoint".Switch_left := FALSE;
	            #"Cmd+Setpoint".Switch_right := FALSE;
	            #"Cmd+Setpoint".Switch_right_to_st := FALSE;
	            #"Cmd+Setpoint".Switch_left_to_st := FALSE;
	        END_IF;
	        
	    END_REGION
	    
	END_REGION
	
	
	
END_FUNCTION_BLOCK
END_NAMESPACE

NAMESPACE Global
FUNCTION_BLOCK FB_VisuAlarm
{ S7_Optimized_Access := 'TRUE' ; Published := 'TRUE' }
VERSION : 0.1
   VAR 
      noAlarmState : Bool;
      CommunicationFault : Struct
         PLC : Word;
         "BW-ASi" : Word;
         Cognex : Word;
         IMC : Word;
         OPC : Word;
      END_STRUCT;
      "BW-ASi" : Struct
         "BW_ASi143 -MCC100 -210KE3 -ConfigErr_Circuit1_Slave(0-15)A_1" : Word;
         "BW_ASi143 -MCC100 -210KE3 -ConfigErr_Circuit1_Slave(16-31)A" : Word;
         "BW_ASi143 -MCC100 -210KE3 -ConfigErr_Circuit1_Slave(0-15)B_1" : Word;
         "BW_ASi143 -MCC100 -210KE3 -ConfigErr_Circuit1_Slave(16-31)B" : Word;
         "BW_ASi143 -MCC100 -210KE3 -PeriErr_Circuit1_Slave(0-15)A_1" : Word;
         "BW_ASi143 -MCC100 -210KE3 -PeriErr_Circuit1_Slave(16-31)A" : Word;
         "BW_ASi143 -MCC100 -210KE3 -PeriErr_Circuit1_Slave(0-15)B_1" : Word;
         "BW_ASi143 -MCC100 -210KE3 -PeriErr_Circuit1_Slave(16-31)B" : Word;
         "BW_ASi143 -MCC100 -210KE3 -ConfigErr_Circuit2_Slave(0-15)A" : Word;
         "BW_ASi143 -MCC100 -210KE3 -ConfigErr_Circuit2_Slave(16-31)A" : Word;
         "BW_ASi143 -MCC100 -210KE3 -ConfigErr_Circuit2_Slave(0-15)B" : Word;
         "BW_ASi143 -MCC100 -210KE3 -ConfigErr_Circuit2_Slave(16-31)B" : Word;
         "BW_ASi143 -MCC100 -210KE3 -PeriErr_Circuit2_Slave(0-15)A" : Word;
         "BW_ASi143 -MCC100 -210KE3 -PeriErr_Circuit2_Slave(16-31)A" : Word;
         "BW_ASi143 -MCC100 -210KE3 -PeriErr_Circuit2_Slave(0-15)B" : Word;
         "BW_ASi143 -MCC100 -210KE3 -PeriErr_Circuit2_Slave(16-31)B" : Word;
         "BW_ASi200 -MCC300 -210KE3 -ConfigErr_Circuit1_Slave(0-15)A" : Word;
         "BW_ASi200 -MCC300 -210KE3 -ConfigErr_Circuit1_Slave(16-31)A" : Word;
         "BW_ASi200 -MCC300 -210KE3 -ConfigErr_Circuit1_Slave(0-15)B" : Word;
         "BW_ASi200 -MCC300 -210KE3 -ConfigErr_Circuit1_Slave(16-31)B" : Word;
         "BW_ASi200 -MCC300 -210KE3 -PeriErr_Circuit1_Slave(0-15)A" : Word;
         "BW_ASi200 -MCC300 -210KE3 -PeriErr_Circuit1_Slave(16-31)A" : Word;
         "BW_ASi200 -MCC300 -210KE3 -PeriErr_Circuit1_Slave(0-15)B" : Word;
         "BW_ASi200 -MCC300 -210KE3 -PeriErr_Circuit1_Slave(16-31)B" : Word;
         "BW_ASi200 -MCC300 -210KE3 -ConfigErr_Circuit2_Slave(0-15)A" : Word;
         "BW_ASi200 -MCC300 -210KE3 -ConfigErr_Circuit2_Slave(16-31)A" : Word;
         "BW_ASi200 -MCC300 -210KE3 -ConfigErr_Circuit2_Slave(0-15)B" : Word;
         "BW_ASi200 -MCC300 -210KE3 -ConfigErr_Circuit2_Slave(16-31)B" : Word;
         "BW_ASi200 -MCC300 -210KE3 -PeriErr_Circuit2_Slave(0-15)A" : Word;
         "BW_ASi200 -MCC300 -210KE3 -PeriErr_Circuit2_Slave(16-31)A" : Word;
         "BW_ASi200 -MCC300 -210KE3 -PeriErr_Circuit2_Slave(0-15)B" : Word;
         "BW_ASi200 -MCC300 -210KE3 -PeriErr_Circuit2_Slave(16-31)B" : Word;
      END_STRUCT;
      "word" : Struct
         Line : Struct
            ProductionLine : Struct
               Conveyor : Array[_.gminProductionLine.._.gmaxProductionLine] of Word;
            END_STRUCT;
            EmptyLine : Struct
               Conveyor : Array[_.gminEmptyLine.._.gmaxEmptyLine] of Word;
            END_STRUCT;
            PackedLine : Struct
               Conveyor : Array[_.gminPackedLine.._.gmaxPackedLine] of Word;
            END_STRUCT;
         END_STRUCT;
      END_STRUCT;
   END_VAR


BEGIN
	// ==========================================================================================================================================
	// Company        : LogTech, s.r.o.
	// Created by     : Mahmoud Elnady
	// Block          : FC_VisuAlarm
	// Project        : Lékárna Chrudim
	// Project number : 23-157
	// ==========================================================================================================================================
	REGION initial state
	    
	    // ESTOP alarm has priority
	    // So, if there are any estop active, other alarms can't be displayed on Alarm screen
	    
	    // no alarm state
	    #noAlarmState :=
	    IDB_GlobalStatus.Line.ProductionLine.Estop OR
	    IDB_GlobalStatus.Line.ProductionLine.Estop OR
	    IDB_GlobalStatus.Line.ProductionLine.Estop;
	    
	    IF #noAlarmState THEN
	        
	        DB_Alarm."BW-ASi" := #"BW-ASi";
	        DB_Alarm.CommunicationFault := #CommunicationFault;
	        DB_Alarm."word" := #word;
	        //"DB_Alarm".CircuitBreaker := #CircuitBreaker;
	        
	    END_IF;
	    
	END_REGION
	
	REGION ASi Config and Peri alarm
	    
	    IF NOT #noAlarmState THEN
	        // ASi gateway: MCC100-bw23: Circuit 1
	        DB_Alarm."BW-ASi"."BW_ASi143 -MCC100 -210KE3 -ConfigErr_Circuit1_Slave(0-15)A" := _."BW_ASi143 -MCC100 -210KE3 -ConfigErr_Circuit1_Slave(0-15)A";
	        DB_Alarm."BW-ASi"."BW_ASi143 -MCC100 -210KE3 -ConfigErr_Circuit1_Slave(16-31)A" := _."BW_ASi143 -MCC100 -210KE3 -ConfigErr_Circuit1_Slave(16-31)A";
	        DB_Alarm."BW-ASi"."BW_ASi143 -MCC100 -210KE3 -ConfigErr_Circuit1_Slave(0-15)B" := _."BW_ASi143 -MCC100 -210KE3 -ConfigErr_Circuit1_Slave(0-15)B";
	        DB_Alarm."BW-ASi"."BW_ASi143 -MCC100 -210KE3 -ConfigErr_Circuit1_Slave(16-31)B" := _."BW_ASi143 -MCC100 -210KE3 -ConfigErr_Circuit1_Slave(16-31)B";
	        DB_Alarm."BW-ASi"."BW_ASi143 -MCC100 -210KE3 -PeriErr_Circuit1_Slave(0-15)A" := _."BW_ASi143 -MCC100 -210KE3 -PeriErr_Circuit1_Slave(0-15)A";
	        DB_Alarm."BW-ASi"."BW_ASi143 -MCC100 -210KE3 -PeriErr_Circuit1_Slave(16-31)A" := _."BW_ASi143 -MCC100 -210KE3 -PeriErr_Circuit1_Slave(16-31)A";
	        DB_Alarm."BW-ASi"."BW_ASi143 -MCC100 -210KE3 -PeriErr_Circuit1_Slave(0-15)B" := _."BW_ASi143 -MCC100 -210KE3 -PeriErr_Circuit1_Slave(0-15)B";
	        DB_Alarm."BW-ASi"."BW_ASi143 -MCC100 -210KE3 -PeriErr_Circuit1_Slave(16-31)B" := _."BW_ASi143 -MCC100 -210KE3 -PeriErr_Circuit1_Slave(16-31)B";
	        // ASi gateway: MCC100-bw23: Circuit 2
	        DB_Alarm."BW-ASi"."BW_ASi143 -MCC100 -210KE3 -ConfigErr_Circuit1_Slave(0-15)A" := _."BW_ASi143 -MCC100 -210KE3 -ConfigErr_Circuit1_Slave(0-15)A";
	        DB_Alarm."BW-ASi"."BW_ASi143 -MCC100 -210KE3 -ConfigErr_Circuit1_Slave(16-31)A" := _."BW_ASi143 -MCC100 -210KE3 -ConfigErr_Circuit1_Slave(16-31)A";
	        DB_Alarm."BW-ASi"."BW_ASi143 -MCC100 -210KE3 -ConfigErr_Circuit1_Slave(0-15)B" := _."BW_ASi143 -MCC100 -210KE3 -ConfigErr_Circuit1_Slave(0-15)B";
	        DB_Alarm."BW-ASi"."BW_ASi143 -MCC100 -210KE3 -ConfigErr_Circuit1_Slave(16-31)B" := _."BW_ASi143 -MCC100 -210KE3 -ConfigErr_Circuit1_Slave(16-31)B";
	        DB_Alarm."BW-ASi"."BW_ASi143 -MCC100 -210KE3 -PeriErr_Circuit1_Slave(0-15)A" := _."BW_ASi143 -MCC100 -210KE3 -PeriErr_Circuit1_Slave(0-15)A";
	        DB_Alarm."BW-ASi"."BW_ASi143 -MCC100 -210KE3 -PeriErr_Circuit1_Slave(16-31)A" := _."BW_ASi143 -MCC100 -210KE3 -PeriErr_Circuit1_Slave(16-31)A";
	        DB_Alarm."BW-ASi"."BW_ASi143 -MCC100 -210KE3 -PeriErr_Circuit1_Slave(0-15)B" := _."BW_ASi143 -MCC100 -210KE3 -PeriErr_Circuit1_Slave(0-15)B";
	        DB_Alarm."BW-ASi"."BW_ASi143 -MCC100 -210KE3 -PeriErr_Circuit1_Slave(16-31)B" := _."BW_ASi143 -MCC100 -210KE3 -PeriErr_Circuit1_Slave(16-31)B";
	        // ASi gateway: MCC300-bw31 : Circuit 1
	        DB_Alarm."BW-ASi"."BW_ASi200 -MCC300 -210KE3 -ConfigErr_Circuit1_Slave(0-15)A" := _."BW_ASi200 -MCC300 -210KE3 -ConfigErr_Circuit1_Slave(0-15)A";
	        DB_Alarm."BW-ASi"."BW_ASi200 -MCC300 -210KE3 -ConfigErr_Circuit1_Slave(16-31)A" := _."BW_ASi200 -MCC300 -210KE3 -ConfigErr_Circuit1_Slave(16-31)A";
	        DB_Alarm."BW-ASi"."BW_ASi200 -MCC300 -210KE3 -ConfigErr_Circuit1_Slave(0-15)B" := _."BW_ASi200 -MCC300 -210KE3 -ConfigErr_Circuit1_Slave(0-15)B";
	        DB_Alarm."BW-ASi"."BW_ASi200 -MCC300 -210KE3 -ConfigErr_Circuit1_Slave(16-31)B" := _."BW_ASi200 -MCC300 -210KE3 -ConfigErr_Circuit1_Slave(16-31)B";
	        DB_Alarm."BW-ASi"."BW_ASi200 -MCC300 -210KE3 -PeriErr_Circuit1_Slave(0-15)A" := _."BW_ASi200 -MCC300 -210KE3 -PeriErr_Circuit1_Slave(0-15)A";
	        DB_Alarm."BW-ASi"."BW_ASi200 -MCC300 -210KE3 -PeriErr_Circuit1_Slave(16-31)A" := _."BW_ASi200 -MCC300 -210KE3 -PeriErr_Circuit1_Slave(16-31)A";
	        DB_Alarm."BW-ASi"."BW_ASi200 -MCC300 -210KE3 -PeriErr_Circuit1_Slave(0-15)B" := _."BW_ASi200 -MCC300 -210KE3 -PeriErr_Circuit1_Slave(0-15)B";
	        DB_Alarm."BW-ASi"."BW_ASi200 -MCC300 -210KE3 -PeriErr_Circuit1_Slave(16-31)B" := _."BW_ASi200 -MCC300 -210KE3 -PeriErr_Circuit1_Slave(16-31)B";
	        // ASi gateway: MCC300-bw31 : Circuit 2
	        DB_Alarm."BW-ASi"."BW_ASi200 -MCC300 -210KE3 -ConfigErr_Circuit2_Slave(0-15)A" := _."BW_ASi200 -MCC300 -210KE3 -ConfigErr_Circuit2_Slave(0-15)A";
	        DB_Alarm."BW-ASi"."BW_ASi200 -MCC300 -210KE3 -ConfigErr_Circuit2_Slave(16-31)A" := _."BW_ASi200 -MCC300 -210KE3 -ConfigErr_Circuit2_Slave(16-31)A";
	        DB_Alarm."BW-ASi"."BW_ASi200 -MCC300 -210KE3 -ConfigErr_Circuit2_Slave(0-15)B" := _."BW_ASi200 -MCC300 -210KE3 -ConfigErr_Circuit2_Slave(0-15)B";
	        DB_Alarm."BW-ASi"."BW_ASi200 -MCC300 -210KE3 -ConfigErr_Circuit2_Slave(16-31)B" := _."BW_ASi200 -MCC300 -210KE3 -ConfigErr_Circuit2_Slave(16-31)B";
	        DB_Alarm."BW-ASi"."BW_ASi200 -MCC300 -210KE3 -PeriErr_Circuit2_Slave(0-15)A" := _."BW_ASi200 -MCC300 -210KE3 -PeriErr_Circuit2_Slave(0-15)A";
	        DB_Alarm."BW-ASi"."BW_ASi200 -MCC300 -210KE3 -PeriErr_Circuit2_Slave(16-31)A" := _."BW_ASi200 -MCC300 -210KE3 -PeriErr_Circuit2_Slave(16-31)A";
	        DB_Alarm."BW-ASi"."BW_ASi200 -MCC300 -210KE3 -PeriErr_Circuit2_Slave(0-15)B" := _."BW_ASi200 -MCC300 -210KE3 -PeriErr_Circuit2_Slave(0-15)B";
	        DB_Alarm."BW-ASi"."BW_ASi200 -MCC300 -210KE3 -PeriErr_Circuit2_Slave(16-31)B" := _."BW_ASi200 -MCC300 -210KE3 -PeriErr_Circuit2_Slave(16-31)B";
	    ELSE
	        // ASi gateway: MCC100-bw23: Circuit 1
	        DB_Alarm."BW-ASi"."BW_ASi143 -MCC100 -210KE3 -ConfigErr_Circuit1_Slave(0-15)A" := 0;
	        DB_Alarm."BW-ASi"."BW_ASi143 -MCC100 -210KE3 -ConfigErr_Circuit1_Slave(16-31)A" := 0;
	        DB_Alarm."BW-ASi"."BW_ASi143 -MCC100 -210KE3 -ConfigErr_Circuit1_Slave(0-15)B" := 0;
	        DB_Alarm."BW-ASi"."BW_ASi143 -MCC100 -210KE3 -ConfigErr_Circuit1_Slave(16-31)B" := 0;
	        DB_Alarm."BW-ASi"."BW_ASi143 -MCC100 -210KE3 -PeriErr_Circuit1_Slave(0-15)A" := 0;
	        DB_Alarm."BW-ASi"."BW_ASi143 -MCC100 -210KE3 -PeriErr_Circuit1_Slave(16-31)A" := 0;
	        DB_Alarm."BW-ASi"."BW_ASi143 -MCC100 -210KE3 -PeriErr_Circuit1_Slave(0-15)B" := 0;
	        DB_Alarm."BW-ASi"."BW_ASi143 -MCC100 -210KE3 -PeriErr_Circuit1_Slave(16-31)B" := 0;
	        // ASi gateway: MCC100-bw23: Circuit 2
	        DB_Alarm."BW-ASi"."BW_ASi143 -MCC100 -210KE3 -ConfigErr_Circuit1_Slave(0-15)A" := 0;
	        DB_Alarm."BW-ASi"."BW_ASi143 -MCC100 -210KE3 -ConfigErr_Circuit1_Slave(16-31)A" := 0;
	        DB_Alarm."BW-ASi"."BW_ASi143 -MCC100 -210KE3 -ConfigErr_Circuit1_Slave(0-15)B" := 0;
	        DB_Alarm."BW-ASi"."BW_ASi143 -MCC100 -210KE3 -ConfigErr_Circuit1_Slave(16-31)B" := 0;
	        DB_Alarm."BW-ASi"."BW_ASi143 -MCC100 -210KE3 -PeriErr_Circuit1_Slave(0-15)A" := 0;
	        DB_Alarm."BW-ASi"."BW_ASi143 -MCC100 -210KE3 -PeriErr_Circuit1_Slave(16-31)A" := 0;
	        DB_Alarm."BW-ASi"."BW_ASi143 -MCC100 -210KE3 -PeriErr_Circuit1_Slave(0-15)B" := 0;
	        DB_Alarm."BW-ASi"."BW_ASi143 -MCC100 -210KE3 -PeriErr_Circuit1_Slave(16-31)B" := 0;
	        // ASi gateway: MCC300-bw31 : Circuit 1
	        DB_Alarm."BW-ASi"."BW_ASi200 -MCC300 -210KE3 -ConfigErr_Circuit1_Slave(0-15)A" := 0;
	        DB_Alarm."BW-ASi"."BW_ASi200 -MCC300 -210KE3 -ConfigErr_Circuit1_Slave(16-31)A" := 0;
	        DB_Alarm."BW-ASi"."BW_ASi200 -MCC300 -210KE3 -ConfigErr_Circuit1_Slave(0-15)B" := 0;
	        DB_Alarm."BW-ASi"."BW_ASi200 -MCC300 -210KE3 -ConfigErr_Circuit1_Slave(16-31)B" := 0;
	        DB_Alarm."BW-ASi"."BW_ASi200 -MCC300 -210KE3 -PeriErr_Circuit1_Slave(0-15)A" := 0;
	        DB_Alarm."BW-ASi"."BW_ASi200 -MCC300 -210KE3 -PeriErr_Circuit1_Slave(16-31)A" := 0;
	        DB_Alarm."BW-ASi"."BW_ASi200 -MCC300 -210KE3 -PeriErr_Circuit1_Slave(0-15)B" := 0;
	        DB_Alarm."BW-ASi"."BW_ASi200 -MCC300 -210KE3 -PeriErr_Circuit1_Slave(16-31)B" := 0;
	        // ASi gateway: MCC300-bw31 : Circuit 2
	        DB_Alarm."BW-ASi"."BW_ASi200 -MCC300 -210KE3 -ConfigErr_Circuit2_Slave(0-15)A" := 0;
	        DB_Alarm."BW-ASi"."BW_ASi200 -MCC300 -210KE3 -ConfigErr_Circuit2_Slave(16-31)A" := 0;
	        DB_Alarm."BW-ASi"."BW_ASi200 -MCC300 -210KE3 -ConfigErr_Circuit2_Slave(0-15)B" := 0;
	        DB_Alarm."BW-ASi"."BW_ASi200 -MCC300 -210KE3 -ConfigErr_Circuit2_Slave(16-31)B" := 0;
	        DB_Alarm."BW-ASi"."BW_ASi200 -MCC300 -210KE3 -PeriErr_Circuit2_Slave(0-15)A" := 0;
	        DB_Alarm."BW-ASi"."BW_ASi200 -MCC300 -210KE3 -PeriErr_Circuit2_Slave(16-31)A" := 0;
	        DB_Alarm."BW-ASi"."BW_ASi200 -MCC300 -210KE3 -PeriErr_Circuit2_Slave(0-15)B" := 0;
	        DB_Alarm."BW-ASi"."BW_ASi200 -MCC300 -210KE3 -PeriErr_Circuit2_Slave(16-31)B" := 0;
	        
	    END_IF;
	    
	END_REGION
	
	REGION Circuit Breaker
	    
	    DB_Alarm.CircuitBreaker.%X0 := NOT _."CircuitBreaker -fb -Zone1-FC1 -MCC001";
	    DB_Alarm.CircuitBreaker.%X1 := NOT  _."CircuitBreaker -fb -Zone1-FC10 -MCC001";
	    DB_Alarm.CircuitBreaker.%X2 := NOT  _."CircuitBreaker -fb -Zone1-FC2 -MCC001";
	    DB_Alarm.CircuitBreaker.%X3 := NOT  _."CircuitBreaker -fb -Zone2-FC1 -MCC001";
	    DB_Alarm.CircuitBreaker.%X4 := NOT  _."CircuitBreaker -fb -Zone2-FC10 -MCC001";
	    DB_Alarm.CircuitBreaker.%X5 := NOT _."CircuitBreaker -fb -Zone2-FC2 -MCC001";
	    DB_Alarm.CircuitBreaker.%X6 := NOT _."CircuitBreaker -fb -Zone2-FC3 -MCC001";
	    
	END_REGION
	
	
	
	
	
END_FUNCTION_BLOCK
END_NAMESPACE

NAMESPACE Global
FUNCTION FC_SafetyAlarm : Void
{ S7_Optimized_Access := 'TRUE' ; Published := 'FALSE' }
VERSION : 0.1

BEGIN
	// ==========================================================================================================================================
	// Company        : LogTech, s.r.o.
	// Created by     : Mahmoud Elnady
	// Block          : FB_Main_LineA1
	// Project        : Lékárna Chrudim
	// Project number : 23-157
	// ==========================================================================================================================================
	
	REGION HMI Alarm
	    
	    DB_Alarm.Estop.%X0 :=
	    _.DB_SafetyStandard.PressReset;
	    DB_Alarm.Estop.%X1 :=
	    _.DB_SafetyStandard.ToStandard.EstopActive;
	    DB_Alarm.Estop.%X2 :=
	    _.DB_SafetyStandard.ToHMI."PhaseOK -MCC001";    
	    DB_Alarm.Estop.%X3 :=
	    _.DB_SafetyStandard.ToHMI."EstopPB -MCC001+SF1";
	    
	END_REGION
END_FUNCTION
END_NAMESPACE

NAMESPACE Global
FUNCTION_BLOCK FB_Merging
{ S7_Optimized_Access := 'TRUE' ; Published := 'TRUE' }
VERSION : 0.1
   VAR_INPUT 
      StraightSensor : Bool;
      ArmSensor : Bool;
   END_VAR

   VAR 
      StraightToteTimer {InstructionName := 'TON_TIME'; LibVersion := '1.0'; S7_SetPoint := 'False'} : TON_TIME;
      ArmToteTimer {InstructionName := 'TON_TIME'; LibVersion := '1.0'} : TON_TIME;
      Priority { ExternalAccessible := 'False'; ExternalVisible := 'False'; ExternalWritable := 'False'} : Struct
         Straight { ExternalAccessible := 'False'; ExternalVisible := 'False'; ExternalWritable := 'False'} : Bool;
         Arm { ExternalAccessible := 'False'; ExternalVisible := 'False'; ExternalWritable := 'False'} : Bool;
      END_STRUCT;
   END_VAR


BEGIN
	// ==========================================================================================================================================
	// Company        : LogTech, s.r.o.
	// Created by     : Anton Vinoth Soundraraj
	// Block          : FB_Merging
	// Project        : LT-Lib-Block
	// ==========================================================================================================================================
	
	REGION PRIORITY MERGING
	    
	    // Priority Check
	    // Occ duration : tote in straight flow
	    #StraightToteTimer(IN := #StraightSensor,
	                       PT := t#24h);
	    // Occ duration : tote from left flow
	    #ArmToteTimer(IN := #ArmSensor,
	                  PT := t#24h);
	    
	    // assign priority
	    // Priority: straight tote
	    IF (#StraightToteTimer.ET >=
	        #ArmToteTimer.ET) THEN
	        #Priority.Straight := TRUE;
	        #Priority.Arm := FALSE;
	    END_IF;
	    // Priority: Arm tote
	    IF (#StraightToteTimer.ET <
	        #ArmToteTimer.ET) THEN
	        #Priority.Straight := FALSE;
	        #Priority.Arm := TRUE;
	    END_IF;
	    
	    // add the priority signals in downstream
	    
	END_REGION
END_FUNCTION_BLOCK
END_NAMESPACE

NAMESPACE Global
FUNCTION_BLOCK FB_SensorBlockage
{ S7_Optimized_Access := 'TRUE' ; Published := 'TRUE' }
VERSION : 0.1
   VAR_INPUT 
      ConveyorSensor : Bool;
      StatusRunning : Bool;
      SensorBlockagePeriod : Time;
   END_VAR

   VAR_OUTPUT 
      SensorBlocked : Bool;
      CurrentBlockageTimerValue : Time;
      ReadBlockageStatus : Bool;
   END_VAR

   VAR 
      SensorBlockageTimer {InstructionName := 'IEC_TIMER'; LibVersion := '1.0'} : IEC_TIMER;
      SensorBlockage { S7_SetPoint := 'True'} : Bool;
      SensorBlockageCondition : Bool;
      FallingEdge {InstructionName := 'F_TRIG'; LibVersion := '1.0'} : F_TRIG;
      FallingEdgeConveyorSensor { S7_SetPoint := 'True'} : Bool;
      BlockageStatus : Bool;
   END_VAR


BEGIN
	// ==========================================================================================================================================================================
	// Company       : LogTech, s.r.o.
	// Created by    : Anton Vinoth Soundraraj
	// Block         : FB_SensorBlockage
	// Project       : LT-Lib-Block
	// ==========================================================================================================================================================================
	
	REGION PEC BLOCKAGE
	    
	    #SensorBlockageCondition :=
	    #StatusRunning AND #ConveyorSensor;
	    
	    // Blockage Timer
	    // !!!! PEC had been blocked for 't' seconds and giving the result as SensorBlockage
	    
	    #SensorBlockageTimer.TON(IN := #SensorBlockageCondition,
	                             PT := #SensorBlockagePeriod,
	                             Q => #SensorBlockage,
	                             ET => #CurrentBlockageTimerValue);
	    
	    IF #SensorBlockage THEN
	        #SensorBlocked := TRUE;
	        #BlockageStatus := TRUE;
	    END_IF;
	    
	END_REGION
	
	REGION Blockage Reset
	    
	    // Can reset the sensor blockage (!!!!!!!) only if the sensor blockage is removed
	    
	    // Falling trigger of the conveyor sensor
	    #FallingEdge(CLK := #ConveyorSensor,
	                 Q => #FallingEdgeConveyorSensor);
	    
	    IF #FallingEdgeConveyorSensor THEN
	        #SensorBlocked := FALSE;
	        #BlockageStatus := FALSE;
	    END_IF;
	    
	    #ReadBlockageStatus := #BlockageStatus;
	    
	END_REGION
	
	
END_FUNCTION_BLOCK
END_NAMESPACE

NAMESPACE Global
FUNCTION_BLOCK DataMan262
{ S7_Optimized_Access := 'TRUE' ; Published := 'FALSE' }
VERSION : 0.1
   VAR_INPUT 
      TriggerSignal : Bool;
      ContinuousGetResults : Bool;
      "Dataman-Results Available" : Bool;
      "Dataman-TriggerReady" : Bool;
      "Dataman-TriggerAck" : Bool;
      "Dataman-Train Focus Ack" : Bool;
      "Dataman-Train Match String Ack" : Bool;
      "Dataman-Execute DMCC Ack" : Bool;
      "Dataman-Set Match String Ack" : Bool;
      "Dataman-ResultID" : Int;
      "Dataman-Result Code" : Int;
      "Dataman-Result Length" : Int;
      "Result Data" : BarCode;
   END_VAR

   VAR_OUTPUT 
      "Dataman-UserData Length" : Word;
      "Dataman-UserData Option" : Word;
      "User Data" : BarCode;
   END_VAR

   VAR_IN_OUT 
      "Dataman-TriggerEnable" : Bool;
      "Dataman-Trigger" : Bool;
      "Dataman-ResultsAck" : Bool;
      "Dataman-Train Focus" : Bool;
      "Dataman-Train Match String" : Bool;
      "Dataman-Execute DMCC" : Bool;
      "Dataman-Set Match String" : Bool;
   END_VAR

   VAR 
      "Result Pending" : Bool;
      "Latest Results" : Struct
         ID : Int;
         Flags : Int;
         Length : Int;
         Value : Array[0..63] of Byte;
      END_STRUCT;
      "Train Focus" : Bool;
      "Train MatchString" : Bool;
      "Execute DMCC" : Bool;
      "Set Match String" : Bool;
      "String" : String[64] := '||>REBOOT$R$L';
      "Match String" : Array[0..63] of Byte;
      "Char" : Array[0..63] of Byte;
      Ret_val_1 { ExternalAccessible := 'False'; ExternalVisible := 'False'; ExternalWritable := 'False'} : Byte;
      R_TRIG_SimpleRead {InstructionName := 'R_TRIG'; LibVersion := '1.0'} : R_TRIG;
      R_TRIG_TrainFocus {InstructionName := 'R_TRIG'; LibVersion := '1.0'} : R_TRIG;
      "R_TRIG_Train MatchString" {InstructionName := 'R_TRIG'; LibVersion := '1.0'} : R_TRIG;
      R_TRIG_ExcuteDMCC {InstructionName := 'R_TRIG'; LibVersion := '1.0'} : R_TRIG;
      R_TRIG_SetMatchString {InstructionName := 'R_TRIG'; LibVersion := '1.0'} : R_TRIG;
      HoldTrigger { S7_SetPoint := 'True'} : Bool;
      HoldTrainFocus : Bool;
      HoldTrainMatchString : Bool;
      HoldDMCCExcute : Bool;
      HoldSetMatchString : Bool;
   END_VAR


BEGIN
	// ==========================================================================================================================================
	// Company        : LogTech, s.r.o.
	// Created by     : Mahmoud Elnady
	// Block          : FC_UpstreaProductionTote
	// Project        : Lekarna, Chrudim -PLC001 -MCC001
	// Project number : 23-157
	// ==========================================================================================================================================
	
	// This block will wait FOR the camera TO become ready, issue a trigger, wait FOR
	//the read TO complete AND THEN copy the read results TO DB5 ("LatestResults").
	//Trigger a read and retrieve the result data.
	REGION Simple Read
	           //Trigger a read and retrieve the result data.      
	    #R_TRIG_SimpleRead(CLK:=#TriggerSignal AND
	                       NOT #ContinuousGetResults);
	    IF #R_TRIG_SimpleRead.Q THEN
	        #HoldTrigger := TRUE;
	    END_IF;
	           
	    IF #HoldTrigger
	           THEN
	               //Make sure triggering is enabled 
	               REGION Triggering is Enabled 
	                   IF NOT #"Dataman-TriggerEnable" THEN
	                       #"Dataman-TriggerEnable" := TRUE;
	                   END_IF;
	               END_REGION
	               
	               //Special case (step 1): If results were already waiting before we issued a 
	               //trigger, process those results before starting a new read sequence.
	               REGION Process Results
	                   IF #"Dataman-Results Available" AND
	                       NOT #"Result Pending"
	                   THEN
	                       #"Result Pending" := TRUE;
	                       #"Dataman-ResultsAck" := TRUE;
	                   END_IF;
	                   
	               END_REGION
	               
	               //If camera ready and trigger not already issued, issue trigger signal. 
	               REGION Trigger Signal
	                   IF #"Dataman-TriggerReady" AND
	                       NOT #"Dataman-Trigger" AND
	                       NOT #"Dataman-TriggerAck" AND
	                       NOT #"Dataman-Results Available" AND
	                       NOT #"Dataman-ResultsAck" AND
	                       NOT #"Result Pending"
	                   THEN
	                       #"Dataman-Trigger" := TRUE;
	                       #"Result Pending" := TRUE;
	                   END_IF;
	                   
	               END_REGION
	               
	               //If results available, get the read results
	               REGION Read results
	                   IF #"Result Pending" AND
	                       #"Dataman-Results Available" AND
	                       NOT #"Dataman-ResultsAck"
	                   THEN
	                       #"Dataman-Trigger" := FALSE;
	                       #"Dataman-ResultsAck" := TRUE;
	                       #"Latest Results".ID := #"Dataman-ResultID";
	                       #"Latest Results".Flags := #"Dataman-Result Code";
	                       #"Latest Results".Length := #"Dataman-Result Length";
	                       MOVE_BLK(IN := #"Result Data"."Result Data"[0],
	                                COUNT := 64,
	                                OUT => #"Latest Results".Value[0]);
	                   END_IF;
	                   
	               END_REGION
	               
	               //Reset trigger signal as soon as it is acknowledged
	               //Reset results acknowledge signal as soon as it is recognized BY the reader.
	               
	               //This is the end OF the read sequence. Reset the "results pending" flag, set the
	               //output TO signal the operation is complete.
	               
	               //Note, the reader signals "results acknowledge" BY setting "results available" TO zero.
	               
	               REGION Reset trigger
	                   
	                   IF #"Result Pending" AND
	                           #"Dataman-ResultsAck" AND
	                           NOT #"Dataman-Results Available"
	                       THEN
	                           #"Dataman-ResultsAck" := FALSE;
	                           #"Result Pending" := FALSE;
	                           #HoldTrigger := FALSE;
	                       END_IF;
	                       
	               END_REGION
	               
	           END_IF;
	       END_REGION
	       
	//Read result data which was triggered elsewhere (i.e. manual trigger button)
	REGION Results Only
	           IF #ContinuousGetResults AND
	               NOT #TriggerSignal
	           THEN
	               
	               //IF results available, save the read results AND issue an acknowledge
	               REGION manual trigger button
	                   IF  #"Dataman-Results Available" AND
	                       NOT #"Dataman-ResultsAck"
	                   THEN
	                       #"Dataman-ResultsAck" := TRUE;
	                       #"Latest Results".ID := #"Dataman-ResultID";
	                       #"Latest Results".Flags := #"Dataman-Result Code";
	                       #"Latest Results".Length := #"Dataman-Result Length";
	                       MOVE_BLK(IN := #"Result Data"."Result Data"[0],
	                                COUNT := 64,
	                                OUT => #"Latest Results".Value[0]);
	                   END_IF;
	                   
	               END_REGION
	               
	               //IF the result acknowledge is complete, reset the result signal
	               REGION Reset signal
	                   IF #"Dataman-ResultsAck" AND
	                       NOT #"Dataman-Results Available"
	                   THEN
	                       #"Dataman-ResultsAck" := FALSE;
	                   END_IF;
	               END_REGION
	           END_IF;
	       END_REGION
	
	//Perform "Train Focus" operation.
	//Note, this operation only enables the training TO occur. After
	//executing this call the reader must be triggered TO perform the actual training.
	
	REGION Train Focus
	    //Perform "Train Focus" operation.
	    #R_TRIG_TrainFocus(CLK:=#"Train Focus");
	    
	    IF #R_TRIG_TrainFocus.Q THEN
	        #HoldTrainFocus := TRUE;
	    END_IF;
	    
	    IF #HoldTrainFocus THEN
	               REGION Initiate the "Train Focus"
	                   //Initiate the "Train Focus" operation AND monitor it TO completion.
	                   IF  NOT #"Dataman-Train Focus" AND
	                       NOT #"Dataman-Train Focus Ack"
	                   THEN
	                       #"Dataman-Train Focus" := True;
	                   END_IF;
	                   
	               END_REGION
	               
	               //Release "Train Focus" signal as soon as it is acknowledged by the reader
	               REGION Release "Train Focus"
	                   
	                   IF #"Dataman-Train Focus Ack" THEN
	                       #"Dataman-Train Focus" := FALSE;
	                       #HoldTrainFocus := FALSE;
	                   END_IF;
	                   
	               END_REGION
	           END_IF;
	       END_REGION
	
	
	//Perform "Train Match String" operation.
	//Note, this operation only enables the training TO occur. After
	//executing this call the reader must be triggered TO perform
	//the actual training.
	
	REGION Train MatchString
	    //Perform "Train Match String" operation.
	    #"R_TRIG_Train MatchString"(CLK:=#"Train MatchString");
	    
	    IF #"R_TRIG_Train MatchString".Q THEN
	        #HoldTrainMatchString := TRUE;
	    END_IF;
	    
	    IF  #HoldTrainMatchString THEN
	       //Issue "Train Match String" signal. 
	       REGION Issue Train Match String
	              IF  NOT #"Dataman-Train Match String" AND
	                       NOT #"Dataman-Train Match String Ack"
	                   THEN
	                       #"Dataman-Train Match String" := TRUE;
	              END_IF;
	       END_REGION
	               
	       //Release "Train Match String" signal as soon as it is acknowledged by the reader.
	       REGION Release "Train Match String"
	              IF #"Dataman-Train Match String Ack" THEN
	                  #"Dataman-Train Match String" := FALSE;
	                  #HoldTrainMatchString := FALSE;
	              END_IF;
	       END_REGION
	   END_IF;
	   
	END_REGION
	
	REGION DMCC Execute
	    //Perform "Execute DMCC" operation.
	    #R_TRIG_ExcuteDMCC(CLK := #"Execute DMCC");
	    
	    IF #R_TRIG_ExcuteDMCC.Q THEN
	        #HoldDMCCExcute := TRUE;
	    END_IF;
	    
	    IF #HoldDMCCExcute THEN
	        //Copy the DMCC command, and then issue the "DMCC Execute" signal.
	        REGION issue the "DMCC Execute"
	            
	            IF  NOT #"Dataman-Execute DMCC" AND
	                NOT #"Dataman-Execute DMCC Ack"
	            THEN
	                #"Dataman-Execute DMCC" := TRUE;
	                #"Dataman-UserData Length" := LEN(#String);
	                
	                Strg_TO_Chars(Strg := #String,
	                              pChars := 0,
	                              Cnt => #"Dataman-UserData Length",
	                              Chars := #"Match String");
	                
	                MOVE_BLK(IN := #"Match String"[0],
	                         COUNT := 64,
	                         OUT => #"User Data"."Result Data"[0]);
	            END_IF;
	            
	        END_REGION
	        
	        //Release "Execute DMCC" signal as soon as it is acknowledged by the reader.
	        REGION Release "Execute DMCC"
	            
	            IF #"Dataman-Execute DMCC Ack" THEN
	                #"Dataman-Execute DMCC" := FALSE;
	                #HoldDMCCExcute := FALSE;
	            END_IF;
	            
	        END_REGION
	    END_IF;
	END_REGION
	
	
	//Perform "Set Match String" operation.
	
	//Set the match String option, copy the Match String value, AND THEN issue "SetMatchString" signal.
	
	//Note, The symbology target's set are selected BY the value OF "UserDataOption".
	//0 = Set all symbologies
	//1 = Set only 2D
	//2 = Set only QR
	//3 = Set only 1D/stacked/postal
	
	REGION Set Match String
	    //Perform "Set Match String" operation.
	    #R_TRIG_SetMatchString(CLK:=#"Set Match String");
	    
	    IF #R_TRIG_SetMatchString.Q THEN
	        #HoldSetMatchString := TRUE;
	    END_IF;
	    
	    IF  #HoldSetMatchString THEN
	        REGION Set the match String option
	            IF NOT #"Dataman-Set Match String" AND
	                NOT #"Dataman-Set Match String Ack"
	            THEN
	                #"Dataman-Set Match String" := TRUE;
	                #"Dataman-UserData Option" := 1;
	                #"Dataman-UserData Length" := LEN(#String);
	                
	                Strg_TO_Chars(Strg := #String,
	                              pChars := 0,
	                              Cnt => #"Dataman-UserData Length",
	                              Chars := #Char);
	                
	                #Ret_val_1 := MOVE_BLK_VARIANT(SRC := #Char[0],
	                                               COUNT := 64,
	                                               SRC_INDEX := 0,
	                                               DEST_INDEX := 0,
	                                               DEST => #"Match String"[0]);
	                
	                MOVE_BLK(IN := #"Match String"[0],
	                         COUNT := 64,
	                         OUT => #"User Data"."Result Data"[0]);
	            END_IF;
	            
	        END_REGION
	        
	        //Release "SetMatchString" signal as soon as it is acknowledged BY the reader.
	        REGION Release "SetMatchString"
	            
	            IF #"Dataman-Set Match String Ack" THEN
	                #"Dataman-Set Match String" := FALSE;
	                #HoldSetMatchString := FALSE;
	            END_IF;
	            
	        END_REGION
	    END_IF;
	END_REGION
	
	
	
	
	
	
END_FUNCTION_BLOCK
END_NAMESPACE

NAMESPACE Global
FUNCTION_BLOCK FB_KlaxonLampYellow
{ S7_Optimized_Access := 'TRUE' ; Published := 'TRUE' }
VERSION : 0.1
   VAR_INPUT 
      BlinkCondition : Bool;
      GlowCondition : Bool;
      BlockageStatus : Bool;
   END_VAR

   VAR_OUTPUT 
      YellowLamp : Bool;
   END_VAR

   VAR 
      Startup {InstructionName := 'IEC_TIMER'; LibVersion := '1.0'; S7_SetPoint := 'False'} : IEC_TIMER;
      StartupActive { S7_SetPoint := 'True'} : Bool;
      AlertTime : Time := T#5s;
      LampGlowON : Bool;
   END_VAR


BEGIN
	// ==========================================================================================================================================================================
	// Company      : LogTech, s.r.o.
	// Created by   : Anton Vinoth Soundraraj
	// Project      : LT-Lib-Block
	// Block        : FB_KlaxonLampYellow
	// ==========================================================================================================================================================================
	
	REGION Lamp Blink
	    
	    // Blink condition System Start
	    // Lamp blink will be active for given preset time
	    
	    #Startup.TOF(IN := #BlinkCondition,
	                 PT := #AlertTime,
	                 Q => #StartupActive);
	    
	END_REGION
	
	REGION Lamp Glow
	    
	    // Lamp will be glowing if glow condition(all conveyors status ready) is set
	    
	    #LampGlowON :=
	    #GlowCondition AND
	    NOT #StartupActive;
	    
	END_REGION
	
	REGION Lamp Glow and Blink
	    
	    // write glow and blink condition to the lamp 
	    
	    #YellowLamp :=
	    #LampGlowON OR
	    (#StartupActive AND
	    _.DB_Sync.ClockBit."Clock_0.5Hz") OR 
	    (#BlockageStatus AND
	    _.DB_Sync.ClockBit."Clock_0.5Hz");
	    
	END_REGION
	
END_FUNCTION_BLOCK
END_NAMESPACE

NAMESPACE EmptyLine
FUNCTION_BLOCK FB_ToggleDir
{ S7_Optimized_Access := 'TRUE' ; Published := 'FALSE' }
VERSION : 0.1
   VAR 
      "J1.5.4" : _.Global.ToggelDir;
      "Toggle_J1.5.4" : Struct
         StarightDir : Bool;
         ArmDir : Bool;
      END_STRUCT;
   END_VAR


BEGIN
	// ==========================================================================================================================================
	// Company        : LogTech, s.r.o.
	// Created by     : Mahmoud Elnady
	// Block          : FB_Toggel Direction
	// Project        : Lekarna, Chrudim -PLC001 -MCC001
	// Project number : 23-157
	// ==========================================================================================================================================
	
	REGION J1.5.4
	    REGION J1.5.4
	        #"J1.5.4"(Sensor := IDB_EmptyLine."J1.5.4".FilteredSensor,
	                  ArmSensor := IDB_EmptyLine."K1.1.1".FilteredSensor,
	                  StraightSensor :=  IDB_EmptyLine."J1.7.1".FilteredSensor,
	                  Toggle => #"Toggle_J1.5.4");
	    END_REGION
	    
	    REGION Straight
	        // Go Straight
	        IF #"Toggle_J1.5.4".StarightDir THEN
	            // Statement section IF
	            ToteDir.Conveyor[_."J1.6.1"].Straight := TRUE;
	            ToteDir.Conveyor[_."J1.6.1"].toRight := FALSE;
	            ToteDir.Conveyor[_."J1.6.1"].toLeft := FALSE;
	        END_IF;
	    END_REGION
	    
	    
	    REGION GoToLeft
	        //Go to the left
	        IF #"Toggle_J1.5.4".ArmDir THEN
	            // Statement section IF
	            ToteDir.Conveyor[_."J1.6.1"].Straight := FALSE;
	            ToteDir.Conveyor[_."J1.6.1"].toRight := FALSE;
	            ToteDir.Conveyor[_."J1.6.1"].toLeft := TRUE;
	        END_IF;
	    END_REGION
	END_REGION
	
	
	
END_FUNCTION_BLOCK
END_NAMESPACE

NAMESPACE Global
FUNCTION_BLOCK ToggelDir
{ S7_Optimized_Access := 'TRUE' ; Published := 'TRUE' }
VERSION : 0.1
   VAR_INPUT 
      Sensor : Bool;
      ArmSensor : Bool;
      StraightSensor : Bool;
   END_VAR

   VAR_OUTPUT 
      Toggle : Struct
         StarightDirection : Bool;
         ArmDirection : Bool;
      END_STRUCT;
   END_VAR

   VAR 
      UpCounter {InstructionName := 'CTU_INT'; LibVersion := '1.0'; S7_SetPoint := 'False'} : CTU_INT;
   END_VAR
   VAR RETAIN
      statResetCounter { S7_SetPoint := 'True'} : Bool;
   END_VAR
   VAR 
      SortAll : Struct
         Staright : Bool;
         Arm : Bool;
      END_STRUCT;
   END_VAR


BEGIN
	// ==========================================================================================================================================
	// Company        : LogTech, s.r.o.
	// Created by     : Mahmoud Elnady
	// Block          : FB_Toggel Direction
	// Project        : Lekarna, Chrudim -PLC001 -MCC001
	// Project number : 23-157
	// ==========================================================================================================================================
	
	// =============================
	// REGION Counter
	// Toggle counter: 0 = Straight, 1 = Arm
	// =============================
	IF #UpCounter.CV >= #UpCounter.PV THEN
	    #statResetCounter := TRUE;
	ELSE
	    #statResetCounter := FALSE;
	END_IF;
	
	#UpCounter(
	           CU := #Sensor,          // input pulse to count
	           R := #statResetCounter, // reset when PV reached
	           PV := 2                 // count up to 2 (0 → 1 → reset)
	);
	
	// =============================
	// REGION SortAll
	// Detect which sensor requests sorting
	// =============================
	#SortAll.Staright := #StraightSensor AND NOT #ArmSensor;
	#SortAll.Arm := #ArmSensor AND NOT #StraightSensor;
	
	// =============================
	// REGION Direction Selection
	// Decide final direction without contradiction
	// =============================
	IF #SortAll.Staright THEN
	    // Straight has priority if its sensor is active
	    #Toggle.StarightDirection := TRUE;
	    #Toggle.ArmDirection := FALSE;
	    
	ELSIF #SortAll.Arm THEN
	    // Arm if its sensor is active
	    #Toggle.StarightDirection := FALSE;
	    #Toggle.ArmDirection := TRUE;
	    
	ELSE
	    // No sensors → fall back to counter toggle
	    IF #UpCounter.CV = 0 THEN
	        #Toggle.StarightDirection := TRUE;
	        #Toggle.ArmDirection := FALSE;
	    ELSE // CV = 1
	        #Toggle.StarightDirection := FALSE;
	        #Toggle.ArmDirection := TRUE;
	    END_IF;
	END_IF;
	
	
	
	
	
	
	
	    
	    
	
	
	
END_FUNCTION_BLOCK
END_NAMESPACE

NAMESPACE Global
FUNCTION_BLOCK FB_EnergySave
{ S7_Optimized_Access := 'TRUE' ; Published := 'TRUE' }
VERSION : 0.1
   VAR_INPUT 
      StatusReady : Bool;
      StatusOccupied : Bool;
      StartUpIN : Bool;
      USOcc : Bool;
      EnergySaveTimePT : Time;
   END_VAR

   VAR_OUTPUT 
      EnergySaveTimeET : Time;
      EnergySaveOut : Bool;
   END_VAR

   VAR 
      EnergySaveTimer {InstructionName := 'IEC_TIMER'; LibVersion := '1.0'} : IEC_TIMER;
      EnergySave { S7_SetPoint := 'True'} : Bool;
   END_VAR


BEGIN
	// ==========================================================================================================================================================================================
	// Company       : LogTech, s.r.o.
	// Created by    : Anton Vinoth Soundraraj
	// Block         : FB_EnergySave
	// Project       : LT-Lib-Block
	// ==========================================================================================================================================================================================
	
	REGION Energy Save
	    
	    // Start energy save timer under certain conditions
	    #EnergySave := NOT #StatusReady OR #StatusOccupied OR #USOcc OR #StartUpIN;
	    
	    // Conveyor running under energy save condition for the preset time which is according to the length of the conveyor
	    #EnergySaveTimer.TOF(IN := #EnergySave,
	                         PT := #EnergySaveTimePT,
	                         Q => #EnergySaveOut,
	                         ET => #EnergySaveTimeET);
	    
	END_REGION
END_FUNCTION_BLOCK
END_NAMESPACE

NAMESPACE Global
FUNCTION_BLOCK FB_RunStop
{ S7_Optimized_Access := 'TRUE' ; Published := 'TRUE' }
VERSION : 0.1
   VAR_INPUT 
      StatusReady : Bool;
      StatusOccu : Bool;
      MotorReverseIN : Bool;
      DSOcc : Bool;
      USOcc : Bool;
      EnergySave : Bool;
      ILStop : Bool;
      PecBlockage : Bool;
   END_VAR

   VAR_OUTPUT 
      MotorForward : Bool;
      MotorReverse : Bool;
   END_VAR

   VAR 
      RunRevIN : Bool;
      RunRev : Bool;
      RunFor : Bool;
   END_VAR


BEGIN
	// ==========================================================================================================================================================================
	// Company       : LogTech, s.r.o.
	// Created by    : Anton Vinoth Soundraraj
	// Block         : FB_RunStop
	// Project       : LT-Lib-Block
	// ==========================================================================================================================================================================
	
	REGION Run/Stop Forward
	    
	    // Run forward
	    #RunFor := #StatusReady AND NOT #MotorReverseIN AND
	    ((#StatusOccu AND NOT #DSOcc) OR (NOT #StatusOccu AND #USOcc)
	    OR #EnergySave) AND NOT #PecBlockage;
	    
	    // Stop forward
	    IF NOT #StatusReady
	        OR (#StatusOccu AND #DSOcc)
	        OR #ILStop OR NOT #EnergySave OR #MotorReverseIN
	        OR #PecBlockage
	    THEN
	        #RunFor := FALSE;
	    END_IF;
	    
	    #MotorForward := #RunFor;
	    
	END_REGION
	
	REGION Run/Stop Reverse
	    
	    // Run reverse 
	    #RunRevIN := #MotorReverseIN;
	    #RunRev := #StatusReady AND #RunRevIN AND NOT #RunFor;
	    
	    // Stop reverse
	    IF NOT #StatusReady AND NOT #RunRevIN THEN
	        #RunRev := FALSE;
	    END_IF;
	    
	    #MotorReverse := #RunRev;
	    
	END_REGION
END_FUNCTION_BLOCK
END_NAMESPACE

NAMESPACE Global
FUNCTION_BLOCK FB_Sensor
{ S7_Optimized_Access := 'TRUE' ; Published := 'TRUE' }
VERSION : 0.1
   VAR_INPUT 
      Sensor : Bool;
      SensorFilterTime : Array[1..2] of Time;   // Filtering time
   END_VAR

   VAR_OUTPUT 
      FilteredSensor : Bool;
   END_VAR

   VAR 
      SensorFilterTimer {InstructionName := 'IEC_TIMER'; LibVersion := '1.0'} : Array[1..2] of IEC_TIMER;
      Filtering : Struct
         Sensor : Bool;
      END_STRUCT;
      Filtered : Struct
         Sensor : Bool;
      END_STRUCT;
      SensorEdge : Struct
         Positive : Bool;
         Negative : Bool;
      END_STRUCT;
      PosEdge {InstructionName := 'R_TRIG'; LibVersion := '1.0'; S7_SetPoint := 'False'} : R_TRIG;
      NegEdge {InstructionName := 'F_TRIG'; LibVersion := '1.0'} : F_TRIG;
   END_VAR


BEGIN
	// ==========================================================================================================================================================================
	// Company       : LogTech, s.r.o.
	// Created by    : Anton Vinoth Soundraraj
	// Block         : FB_Sensor
	// Project       : LT-Lib-Block
	// ==========================================================================================================================================================================
	
	REGION Sensor Filter
	    
	    // Filter timer 1 sending the sensor active signal to the process after preset time
	    #SensorFilterTimer[1].TON(IN := #Sensor,
	                              PT := #SensorFilterTime[1],
	                              Q => #Filtering.Sensor);
	    
	    // Filter timer 2 stop the sensor active signal from the process after preset time
	    #SensorFilterTimer[2].TOF(IN := #Filtering.Sensor,
	                              PT := #SensorFilterTime[2],
	                              Q => #Filtered.Sensor);
	    
	    // Static to output
	    #FilteredSensor := #Filtered.Sensor;
	    
	END_REGION
	
	REGION Sensor Edge Detection
	    
	    #PosEdge(CLK := #Filtered.Sensor);
	    #NegEdge(CLK := #Sensor);
	    #SensorEdge.Positive := #PosEdge.Q;
	    #SensorEdge.Negative := #NegEdge.Q;
	    
	END_REGION
	
END_FUNCTION_BLOCK
END_NAMESPACE

NAMESPACE Global
FUNCTION_BLOCK FB_Klaxon
{ S7_Optimized_Access := 'TRUE' ; Published := 'TRUE' }
VERSION : 0.1
   VAR_INPUT 
      SystemStart : Bool;
      SystemStop : Bool;
      ReadGlobalFault : Bool;
      ReadGlobalReady : Bool;
      ReadEstopActive : Bool;
      ReadGlobalBlockage : Bool;
   END_VAR

   VAR 
      KLAXON_HORN : FB_KlaxonHorn;
      KLAXON_YELLOW : FB_KlaxonLampYellow;
      HORN : Bool;
      YELLOW : Bool;
      GREEN : Bool;
   END_VAR


BEGIN
	// ==========================================================================================================================================================================
	// Company       : LogTech, s.r.o.
	// Created by    : Anton Vinoth Soundraraj
	// Block         : FB_Klaxon
	// Project       : LT-LIB-Block
	// ==========================================================================================================================================================================
	
	REGION Klaxon Horn
	    
	    // FB_KlaxonHorn
	    // Called as MIDB
	    
	    #KLAXON_HORN(Start          := #SystemStart,
	                 Stop           := #SystemStop,
	                 GlobalFault    := #ReadGlobalFault,
	                 GlobalBlockage := #ReadGlobalBlockage,
	                 EstopActive    := #ReadEstopActive,
	                 HornActive     => #HORN);
	    
	END_REGION
	
	REGION Klaxon Yellow
	    
	    // FB_KlaxonLampYellow
	    // Called as MIDB
	    
	    #KLAXON_YELLOW(BlinkCondition := #SystemStart,
	                   GlowCondition  := NOT #ReadGlobalReady,
	                   BlockageStatus := #ReadGlobalBlockage,
	                   YellowLamp     => #YELLOW);
	    
	END_REGION
	
	REGION Klaxon Green
	    
	    #GREEN :=
	    #ReadGlobalReady AND
	    NOT #ReadGlobalBlockage AND
	    NOT #KLAXON_YELLOW.StartupActive AND 
	    NOT #KLAXON_YELLOW.YellowLamp;
	    
	END_REGION
END_FUNCTION_BLOCK
END_NAMESPACE

NAMESPACE Global
FUNCTION_BLOCK FB_KlaxonHorn
{ S7_Optimized_Access := 'TRUE' ; Published := 'TRUE' }
VERSION : 0.1
   VAR_INPUT 
      Start : Bool;
      Stop : Bool;
      GlobalFault : Bool;
      GlobalBlockage : Bool;
      EstopActive : Bool;
      Fire : Bool;
   END_VAR

   VAR_OUTPUT 
      HornActive : Bool;
   END_VAR

   VAR 
      RT_Start {InstructionName := 'R_TRIG'; LibVersion := '1.0'; S7_SetPoint := 'False'} : R_TRIG;
      RT_Stop {InstructionName := 'R_TRIG'; LibVersion := '1.0'} : R_TRIG;
      RT_Estop {InstructionName := 'R_TRIG'; LibVersion := '1.0'} : R_TRIG;
      RT_Fault {InstructionName := 'R_TRIG'; LibVersion := '1.0'} : R_TRIG;
      RT_Blockage {InstructionName := 'R_TRIG'; LibVersion := '1.0'} : R_TRIG;
      RT_Fire {InstructionName := 'R_TRIG'; LibVersion := '1.0'} : R_TRIG;
      KlaxonHornTimer {InstructionName := 'IEC_TIMER'; LibVersion := '1.0'; S7_SetPoint := 'False'} : IEC_TIMER;
      KlaxonHornCondition { S7_SetPoint := 'True'} : Bool;
      HornCondition : Bool;
   END_VAR


BEGIN
	// ==========================================================================================================================================================================
	// Company      : LogTech, s.r.o.
	// Created by   : Anton Vinoth Soundraraj
	// Project      : LT-Lib-Block
	// Block        : FB_KlaxonHorn
	// ==========================================================================================================================================================================
	
	REGION Horn
	    
